(* IEC 61131-3 sources: std_i2980_v2.06_cp053/Source/IMM/ieccontrol/AutoCalibration1 (part 4) *)

GO_ON_TRANSITION TResetCalibBwd (* TResetCalibBwd *) FROM S_StopCalibBwd TO S_RESET :=  #BEGIN_EDIT_BLOCK
TRUE
;#END_EDIT_BLOCK
END_TRANSITION

TRANSITION TStartWriteBwd (* TStartWriteBwd *) FROM S_CHECK_ALARMS_BWD TO S_WRITE_BWD :=  #BEGIN_EDIT_BLOCK
S_CHECK_ALARMS_BWD.T > T#100ms
;#END_EDIT_BLOCK
END_TRANSITION

GO_ON_TRANSITION TStopIdentBwd2 (* TStopCalibBwd2 *) FROM S_CHECK_ALARMS_BWD TO S_StopCalibBwd :=  #BEGIN_EDIT_BLOCK
sv_iPendingAlarms <> 0
;#END_EDIT_BLOCK
END_TRANSITION

TRANSITION TWriteBwd (* TWriteBwd *) FROM S_WRITE_BWD TO S_CHECK_MINSPEED_BWD :=  #BEGIN_EDIT_BLOCK
mbLogFileSaved
;#END_EDIT_BLOCK
END_TRANSITION

TRANSITION TMaxBwdDetected (* TMaxBwdDetected *) FROM S_CHECK_MINSPEED_BWD TO S_MoveEndBwd :=  #BEGIN_EDIT_BLOCK
bMinBwdDetected
;#END_EDIT_BLOCK
END_TRANSITION

TRANSITION TMaxBwdRetry (* TMaxBwdRetry *) FROM S_CHECK_MINSPEED_BWD TO S_ReadyMinBwdRetry :=  #BEGIN_EDIT_BLOCK
bMinBwdRetry
;#END_EDIT_BLOCK
END_TRANSITION

TRANSITION TReadyMinBwdRetry (* Trans49 *) FROM S_ReadyMinBwdRetry TO S_MinBwdRetry :=  #BEGIN_EDIT_BLOCK
fbCheckReady.bReady
;#END_EDIT_BLOCK
END_TRANSITION

TRANSITION TMoveFwdDone (* TMoveFwdDone *) FROM S_MinBwdRetry TO S_CHECK_ALARMS_RETRYBWD :=  #BEGIN_EDIT_BLOCK
bMoveFwdDone
;#END_EDIT_BLOCK
END_TRANSITION

GO_ON_TRANSITION TStopMoveFwd (* TStopMoveFwd *) FROM S_MinBwdRetry TO S_StopMoveFwd :=  #BEGIN_EDIT_BLOCK
sv_GlobalIdentMinSpeedStatus.Status = tnCalibState_Aborted OR
sv_GlobalIdentMinSpeedStatus.Status = tnCalibState_None
OR sv_iPendingAlarms <> 0
OR mActMovement^.bRedo = FALSE

;#END_EDIT_BLOCK
END_TRANSITION

TRANSITION TResetBwd (* TResetBwd *) FROM S_StopMoveFwd TO S_RESET :=  #BEGIN_EDIT_BLOCK
TRUE
;#END_EDIT_BLOCK
END_TRANSITION

TRANSITION TRetryBwd (* TRetryBwd *) FROM S_CHECK_ALARMS_RETRYBWD TO S_CALIB_BWD :=  #BEGIN_EDIT_BLOCK
S_CHECK_ALARMS_RETRYBWD.T > T#1s
;#END_EDIT_BLOCK
END_TRANSITION

GO_ON_TRANSITION TStopIdentBwd4 (* TStopIdentBwd4 *) FROM S_CHECK_ALARMS_RETRYBWD TO S_StopMoveFwd :=  #BEGIN_EDIT_BLOCK
sv_iPendingAlarms <> 0
;#END_EDIT_BLOCK
END_TRANSITION

TRANSITION TMoveEndBwdDone (* TMoveEndBwdDone *) FROM S_MoveEndBwd TO S_Done :=  #BEGIN_EDIT_BLOCK
bMoveBwdDone
;#END_EDIT_BLOCK
END_TRANSITION

GO_ON_TRANSITION TStopMoveEndBwd (* TStopMoveEndBwd *) FROM S_MoveEndBwd TO S_StopMoveEndBwd :=  #BEGIN_EDIT_BLOCK
sv_GlobalIdentMinSpeedStatus.Status = tnCalibState_Aborted OR
sv_GlobalIdentMinSpeedStatus.Status = tnCalibState_None
OR sv_iPendingAlarms <> 0
;#END_EDIT_BLOCK
END_TRANSITION

GO_ON_TRANSITION TResetMoveEndBwd (* TResetMoveEndBwd *) FROM S_StopMoveEndBwd TO S_RESET :=  #BEGIN_EDIT_BLOCK
TRUE
;#END_EDIT_BLOCK
END_TRANSITION

TRANSITION TDone (* TDone *) FROM S_Done TO S_RESET :=  #BEGIN_EDIT_BLOCK
TRUE
;#END_EDIT_BLOCK
END_TRANSITION

(* end IecGraph-Code *)
(* sfc-code *)
(* end sfc-code *)

END_ALGORITHM

POSTUPDATE_ALGORITHM pMinCommandListen ON PU_Task_7 WITH sv_GlobalIdentMinSpeedStatus.Command,sv_GlobalIdentMinSpeedStatus.bStart

VAR_TEMP
 i : DINT;
END_VAR
#BEGIN_EDIT_BLOCK
//stop all calibrations
// TEST
IF sv_GlobalIdentMinSpeedStatus.Command = tnCalibCommand_Stop THEN
    sv_GlobalIdentMinSpeedStatus.bStart := FALSE;
END_IF;
//
IF sv_GlobalIdentMinSpeedStatus.Command = tnCalibCommand_Stop OR (NOT sv_GlobalIdentMinSpeedStatus.bStart) THEN
    FOR i:= 1 TO cCalibMovements DO
        IF CHECK_REF(sv_GlobalIdentMinSpeedStatus.pMovements[i]^) THEN
            IF sv_GlobalIdentMinSpeedStatus.pMovements[i]^.Status = tnCalibState_Running OR
               sv_GlobalIdentMinSpeedStatus.pMovements[i]^.bRedo THEN
                sv_GlobalIdentMinSpeedStatus.pMovements[i]^.Status := tnCalibState_Aborted;
                sv_GlobalIdentMinSpeedStatus.pMovements[i]^.bRedo := FALSE;//FIXME: check if needed
                sv_GlobalIdentMinSpeedStatus.Status := tnCalibState_Aborted;
                EXIT;
            END_IF;
        END_IF;
    END_FOR;
    IF (sv_GlobalIdentMinSpeedStatus.Command = tnCalibCommand_Stop) THEN
       IF (sv_GlobalIdentMinSpeedStatus.Status <> tnCalibState_Aborted) THEN
          sv_GlobalIdentMinSpeedStatus.Status := tnCalibState_None;
       END_IF;

    END_IF;
ELSIF (sv_GlobalIdentMinSpeedStatus.Command = tnCalibCommand_Start) OR (sv_GlobalIdentMinSpeedStatus.bStart) THEN
    IF sv_OperationMode = nSetup THEN
        mbUseSingleMovement := FALSE;
        START_PROCESS_ALGORITHM(paMinCalibSequence);
    ELSE
        sv_GlobalIdentMinSpeedStatus.bStart := FALSE;
        SET_ALARM(erSetupModeRequiredForCalib);
    END_IF;
END_IF;
sv_GlobalIdentMinSpeedStatus.Command := tnCalibCommand_None;

;#END_EDIT_BLOCK END_ALGORITHM

(*
Coordinate sequential start of auto calib cycle
starts one auto calib movement after the other
*)

PROCESS_ALGORITHM paMinCalibSequence ON TaskMid

VAR_TEMP
 j : DINT;
 i : DINT;
END_VAR

VAR
 tmpMovements : tyIdentSpeedMovements;
 iMaxMovements : DINT;
 tmpM : tpIdentSpeedMovement;
 ConstBwdVis : tsVelPre;
END_VAR

(* IecGraph-Code *)

(* init step *)
INITIAL_STEP S_INIT:
ASortCalibs (P);
Action108 (P);
END_STEP

ACTION ASortCalibs: #BEGIN_EDIT_BLOCK
sv_GlobalIdentMinSpeedStatus.Status := tnCalibState_Running;
miErrorNo := 0;

tmpMovements := sv_GlobalIdentMinSpeedStatus.pMovements;

(* get number of movements *)
FOR i:= 1 TO cCalibMovements DO
    IF NOT CHECK_REF(tmpMovements[i]^)  THEN
        EXIT;
    END_IF;
END_FOR;
iMaxMovements := i -1;

(* sort them by iOrder *)
FOR i := 1 TO iMaxMovements -1 DO
    FOR j := 1 TO iMaxMovements - 1 - i +1 DO
        IF tmpMovements[j]^.iOrder > tmpMovements[j + 1]^.iOrder THEN
            tmpM := tmpMovements[j];
            tmpMovements[j] := tmpMovements[j + 1];
            tmpMovements[j + 1] := tmpM;
        END_IF;
    END_FOR;
END_FOR;

;#END_EDIT_BLOCK END_ACTION (*ASortCalibs*)
ACTION Action108: #BEGIN_EDIT_BLOCK
mCalibCounter := 0;
sv_GlobalIdentMinSpeedStatus.iCurrentStep := mCalibCounter;

;#END_EDIT_BLOCK END_ACTION (*Action108*)

(* steps *)
STEP S_RESET:
AReset (P);
AStopMovements (N);
AStopSelf (P);
END_STEP

ACTION AReset: #BEGIN_EDIT_BLOCK
sv_bAutoIdentRunning := FALSE;

;#END_EDIT_BLOCK END_ACTION (*AReset*)
ACTION AStopMovements: #BEGIN_EDIT_BLOCK
(* stop all identification movements *)
FOR i:= 1 TO cCalibMovements DO
    IF CHECK_REF(sv_GlobalIdentMinSpeedStatus.pMovements[i]^) THEN
        IF sv_GlobalIdentMinSpeedStatus.pMovements[i]^.Status = tnCalibState_Running OR
           sv_GlobalIdentMinSpeedStatus.pMovements[i]^.bRedo THEN
            sv_GlobalIdentMinSpeedStatus.pMovements[i]^.Status := tnCalibState_Aborted;
            sv_GlobalIdentMinSpeedStatus.pMovements[i]^.bRedo := FALSE;//FIXME: check if needed
            EXIT;
        END_IF;
    END_IF;
END_FOR;

;#END_EDIT_BLOCK END_ACTION (*AStopMovements*)
ACTION AStopSelf: #BEGIN_EDIT_BLOCK
sv_GlobalIdentMinSpeedStatus.bStart := FALSE;
STOP_PROCESS_ALGORITHM();

;#END_EDIT_BLOCK END_ACTION (*AStopSelf*)
STEP Step74:
AAnyCoreActive (N);
END_STEP

STEP Step19:
ASignalStart (P);
END_STEP

ACTION ASignalStart: #BEGIN_EDIT_BLOCK
sv_bAutoIdentRunning := TRUE;

;#END_EDIT_BLOCK END_ACTION (*ASignalStart*)
STEP S_MoveEjectorBack:
AEjectorBack (P);
Action116 (N);
AResetEjectorBack (P0);
END_STEP

ACTION Action116: #BEGIN_EDIT_BLOCK
fbCheckReady(DeviceId := DeviceIdEjector)

;#END_EDIT_BLOCK END_ACTION (*Action116*)
ACTION AResetEjectorBack: #BEGIN_EDIT_BLOCK
miErrorNo := 0;
sv_EjectorIdentMinMovement.prIdentPosition^ := 0.0;
sv_EjectorIdentMinMovement.prStopRamp^ := 0.0;
sv_EjectorIdentMinMovement.pbMoveIdent^ := FALSE;
sv_EjectorIdentMinMovement.pConstBwdVis^ := ConstBwdVis;

;#END_EDIT_BLOCK END_ACTION (*AResetEjectorBack*)
STEP S_StopEjector:
AStopEjeMovement (P);
END_STEP

STEP S_MoveMoldBack:
AMoldBack (P);
Action118 (N);
AResetMoldBack (P0);
END_STEP

ACTION Action118: #BEGIN_EDIT_BLOCK
fbCheckReady(DeviceId := DeviceIdMold)

;#END_EDIT_BLOCK END_ACTION (*Action118*)
ACTION AResetMoldBack: #BEGIN_EDIT_BLOCK
miErrorNo := 0;
sv_MoldIdentMinMovement.prIdentPosition^ := 0.0;
sv_MoldIdentMinMovement.prStopRamp^ := 0.0;
sv_MoldIdentMinMovement.pbMoveIdent^ := FALSE;
sv_MoldIdentMinMovement.pConstBwdVis^ := ConstBwdVis;

;#END_EDIT_BLOCK END_ACTION (*AResetMoldBack*)
STEP S_StopMold:
AStopMoldMovement (P);
END_STEP

STEP S_CALIB_SINGLE:
AStartMovementStart (P);
END_STEP

ACTION AStartMovementStart: #BEGIN_EDIT_BLOCK
IF mCalibCounter < iMaxMovements THEN
   mCalibCounter := mCalibCounter +1;
   tmpMovements[mCalibCounter]^.bRedo := TRUE;
END_IF;

;#END_EDIT_BLOCK END_ACTION (*AStartMovementStart*)
STEP S_CHECKNEXT:
END_STEP

STEP S_StopIdent:
AStopIdent (P);
END_STEP

ACTION AStopIdent: #BEGIN_EDIT_BLOCK
sv_GlobalIdentMinSpeedStatus.Status := tnCalibState_Done;

;#END_EDIT_BLOCK END_ACTION (*AStopIdent*)

(* transitions *)
TRANSITION Trans50 (* Trans50 *) FROM S_RESET TO S_INIT :=  #BEGIN_EDIT_BLOCK
TRUE
;#END_EDIT_BLOCK
END_TRANSITION

TRANSITION Trans80 (* Trans80 *) FROM S_INIT TO Step19 :=  #BEGIN_EDIT_BLOCK
NOT sv_bCoresActive AND
sv_iPendingAlarms = 0
;#END_EDIT_BLOCK
(*Comment : Start with moving ejector and
mold in backward position, check if any failure
occured.
After that start the calibration cycle, if no alarm is
pending*)
END_TRANSITION

GO_ON_TRANSITION Trans87 (* Trans87 *) FROM S_INIT TO Step74 :=  #BEGIN_EDIT_BLOCK
sv_bCoresActive OR
sv_iPendingAlarms > 0

;#END_EDIT_BLOCK
END_TRANSITION

TRANSITION Trans88 (* Trans88 *) FROM Step74 TO S_RESET :=  #BEGIN_EDIT_BLOCK
TRUE

;#END_EDIT_BLOCK
END_TRANSITION

TRANSITION Trans18 (* Trans18 *) FROM Step19 TO S_MoveEjectorBack :=  #BEGIN_EDIT_BLOCK
TRUE
;#END_EDIT_BLOCK
END_TRANSITION

TRANSITION Trans72 (* Trans72 *) FROM S_MoveEjectorBack TO S_MoveMoldBack :=  #BEGIN_EDIT_BLOCK
fbCheckReady.bReady AND
sv_iPendingAlarms = 0
;#END_EDIT_BLOCK
END_TRANSITION

GO_ON_TRANSITION Trans83 (* Trans83 *) FROM S_MoveEjectorBack TO S_StopEjector :=  #BEGIN_EDIT_BLOCK
sv_GlobalIdentMinSpeedStatus.Status = tnCalibState_Aborted OR
sv_GlobalIdentMinSpeedStatus.Status = tnCalibState_None
OR sv_iPendingAlarms <> 0
;#END_EDIT_BLOCK
END_TRANSITION

TRANSITION Trans84 (* Trans84 *) FROM S_StopEjector TO S_RESET :=  #BEGIN_EDIT_BLOCK
TRUE

;#END_EDIT_BLOCK
END_TRANSITION

TRANSITION Trans81 (* Trans81 *) FROM S_MoveMoldBack TO S_CALIB_SINGLE :=  #BEGIN_EDIT_BLOCK
fbCheckReady.bReady AND
sv_iPendingAlarms = 0
;#END_EDIT_BLOCK
END_TRANSITION

GO_ON_TRANSITION Trans85 (* Trans85 *) FROM S_MoveMoldBack TO S_StopMold :=  #BEGIN_EDIT_BLOCK
sv_GlobalIdentMinSpeedStatus.Status = tnCalibState_Aborted OR
sv_GlobalIdentMinSpeedStatus.Status = tnCalibState_None
OR sv_iPendingAlarms <> 0
;#END_EDIT_BLOCK
END_TRANSITION

TRANSITION Trans86 (* Trans86 *) FROM S_StopMold TO S_RESET :=  #BEGIN_EDIT_BLOCK
TRUE
;#END_EDIT_BLOCK
END_TRANSITION

TRANSITION TCheckActMoveReady (* TCheckActMoveReady *) FROM S_CALIB_SINGLE TO S_CHECKNEXT :=  #BEGIN_EDIT_BLOCK
tmpMovements[mCalibCounter]^.bRedo = FALSE AND
NOT(sv_GlobalIdentMinSpeedStatus.Status = tnCalibState_Aborted OR
    sv_GlobalIdentMinSpeedStatus.Status = tnCalibState_Error)
;#END_EDIT_BLOCK
END_TRANSITION

GO_ON_TRANSITION TCheckError (* TCheckError *) FROM S_CALIB_SINGLE TO S_RESET :=  #BEGIN_EDIT_BLOCK
sv_GlobalIdentMinSpeedStatus.Status = tnCalibState_Aborted OR
sv_GlobalIdentMinSpeedStatus.Status = tnCalibState_Error OR
iMaxMovements = 0
;#END_EDIT_BLOCK
END_TRANSITION

TRANSITION TNextUnit (* TNextUnit *) FROM S_CHECKNEXT TO S_CALIB_SINGLE :=  #BEGIN_EDIT_BLOCK
mCalibCounter < iMaxMovements
//AND S_CHECKNEXT.T>T#3s
;#END_EDIT_BLOCK
END_TRANSITION

TRANSITION TStopIdent (* TStopIdent *) FROM S_CHECKNEXT TO S_StopIdent :=  #BEGIN_EDIT_BLOCK
mCalibCounter >= iMaxMovements
;#END_EDIT_BLOCK
END_TRANSITION

TRANSITION TReset (* TReset *) FROM S_StopIdent TO S_RESET :=  #BEGIN_EDIT_BLOCK
TRUE
;#END_EDIT_BLOCK
END_TRANSITION

(* end IecGraph-Code *)
(* sfc-code *)

(* stand alone actions *)
ACTION AEjectorBack: #BEGIN_EDIT_BLOCK
miErrorNo := cIdentSpeedMinSequence;

IF sv_EjectorIdentMinMovement.bPositionIncreasingFwd THEN
   sv_EjectorIdentMinMovement.prIdentPosition^ := mrBwdStopPosition;
ELSE
   sv_EjectorIdentMinMovement.prIdentPosition^ := sv_EjectorIdentMinMovement.prStroke^ - mrBwdStopPosition;
END_IF;
sv_EjectorIdentMinMovement.prStopRamp^ := 1.0e10;
ConstBwdVis := sv_EjectorIdentMinMovement.pConstBwdVis^;
sv_EjectorIdentMinMovement.pConstBwdVis^.Pressure.Output.rRamp := MAX(1.0e10, sv_EjectorIdentMinMovement.pConstBwdVis^.Pressure.Output.rRamp);
sv_EjectorIdentMinMovement.pConstBwdVis^.Pressure.rMinOutput := 0.1 * sv_EjectorIdentMinMovement.prMaxPressureBwd^;
sv_EjectorIdentMinMovement.pbMoveIdent^ := TRUE;

evStartRequestData.DeviceId := DeviceIdEjector;
evStartRequestData.MoveDir := cMoveBwd;
evStartRequestData.MoveId := cMoveBwd;
SET_EVENT(evStartRequest, evStartRequestData);

;#END_EDIT_BLOCK END_ACTION (*AEjectorBack*)
ACTION AMoldBack: #BEGIN_EDIT_BLOCK
miErrorNo := cIdentSpeedMinSequence;

IF sv_MoldIdentMinMovement.bPositionIncreasingFwd THEN
   sv_MoldIdentMinMovement.prIdentPosition^ := mrBwdStopPosition;
ELSE
   sv_MoldIdentMinMovement.prIdentPosition^ := sv_MoldIdentMinMovement.prStroke^ - mrBwdStopPosition;
END_IF;
sv_MoldIdentMinMovement.prStopRamp^ := 1.0e10;
ConstBwdVis := sv_MoldIdentMinMovement.pConstBwdVis^;
sv_MoldIdentMinMovement.pConstBwdVis^.Pressure.Output.rRamp := MAX(1.0e10, sv_MoldIdentMinMovement.pConstBwdVis^.Pressure.Output.rRamp);
sv_MoldIdentMinMovement.pConstBwdVis^.Pressure.rMinOutput := 0.1 * sv_MoldIdentMinMovement.prMaxPressureBwd^;
sv_MoldIdentMinMovement.pbMoveIdent^ := TRUE;

evStartRequestData.DeviceId := DeviceIdMold;
evStartRequestData.MoveDir := cMoveBwd;
evStartRequestData.MoveId := cMoveBwd;
SET_EVENT(evStartRequest, evStartRequestData);

;#END_EDIT_BLOCK END_ACTION (*AMoldBack*)
ACTION AStopEjeMovement: #BEGIN_EDIT_BLOCK
evStopRequestData.DeviceId := DeviceIdEjector;
evStopRequestData.MoveDir := cMoveBwd;
evStopRequestData.MoveId := cMoveBwd;
SET_EVENT(evStopRequest, evStopRequestData);
IF sv_GlobalIdentMinSpeedStatus.Status <> tnCalibState_None THEN
    sv_GlobalIdentMinSpeedStatus.Status := tnCalibState_Aborted;
END_IF;

;#END_EDIT_BLOCK END_ACTION (*AStopEjeMovement*)
ACTION AStopMoldMovement: #BEGIN_EDIT_BLOCK
evStopRequestData.DeviceId := DeviceIdMold;
evStopRequestData.MoveDir := cMoveBwd;
evStopRequestData.MoveId := cMoveBwd;
SET_EVENT(evStopRequest, evStopRequestData);
IF sv_GlobalIdentMinSpeedStatus.Status <> tnCalibState_None THEN
    sv_GlobalIdentMinSpeedStatus.Status := tnCalibState_Aborted;
END_IF;

;#END_EDIT_BLOCK END_ACTION (*AStopMoldMovement*)
ACTION AAnyCoreActive: #BEGIN_EDIT_BLOCK
IF sv_bCoresActive THEN
   SET_ALARM(erCalibCoresActive);
END_IF;
sv_GlobalIdentMinSpeedStatus.Status := tnCalibState_Aborted;

;#END_EDIT_BLOCK END_ACTION (*AAnyCoreActive*)

(* exits *)

EXIT_TRANSITION E_NotSetupMode := #BEGIN_EDIT_BLOCK
sv_OperationMode <> nSetup
;#END_EDIT_BLOCK
PRIORITY 1 WITH  INITIAL_STEP S_RESET: END_STEP
END_TRANSITION
(* end sfc-code *)

END_ALGORITHM

POSTUPDATE_ALGORITHM pDataState ON PU_Task_13 WITH sv_DataState

VAR_TEMP
 i : DINT;
END_VAR

VAR
 bMDLoadingInProgress : BOOL (* loading of machine data in progress *);
END_VAR
#BEGIN_EDIT_BLOCK
(**************************************** WARNING ********************************************
 *** The KEBA Kemro K2 System including software is not intended for safety control tasks! ***
 ***                       For further information see Comment tab!                        ***
 *********************************************************************************************)

//reset calib state after loading machine data

IF sv_DataState = nReadMachineData THEN
   //loading of machinedata in progress
   bMDLoadingInProgress := TRUE;
   RETURN;
END_IF;

IF sv_DataState = nReady AND bMDLoadingInProgress THEN
   FOR i := 1 TO sv_GlobalIdentMaxSpeedStatus.iMaxStep DO
      //set state to tnCalibState_None
      sv_GlobalIdentMaxSpeedStatus.pMovements[i]^.Status := tnCalibState_None;
   END_FOR;
   FOR i := 1 TO sv_GlobalIdentMinSpeedStatus.iMaxStep DO
      //set state to tnCalibState_None
      sv_GlobalIdentMinSpeedStatus.pMovements[i]^.Status := tnCalibState_None;
   END_FOR;
   bMDLoadingInProgress := FALSE;
END_IF;

;#END_EDIT_BLOCK END_ALGORITHM

END_ALGORITHM_BLOCK

#END_OF_IEC_PART

@Puma @IecEditor 6 152 @Pou 25
@@@BEG_Comment@@@

@@@END_Comment@@@

@BEG_Contents

@BEG_Func
@RT(17)FuncTreeContainer
4
@Var @RT(14)GET_SYNC_REFTO @RT(0) @T @T @DERIVED 0 @F @RT(22)KEBA_STANDARD_FUNCTION @F
@T
@BEG_Attrib
0 @RT(0) @RT(0)
@END_Attrib
1 1 @F @F @F @F

@Var @RT(9)SET_ALARM @RT(0) @T @T @DERIVED 0 @F @RT(23)KEBA_STANDARD_PROCEDURE @F
@T
@BEG_Attrib
0 @RT(0) @RT(0)
@END_Attrib
1 1 @F @F @F @F

@Var @RT(9)SET_EVENT @RT(0) @T @T @DERIVED 0 @F @RT(23)KEBA_STANDARD_PROCEDURE @F
@T
@BEG_Attrib
0 @RT(0) @RT(0)
@END_Attrib
1 1 @F @F @F @F

@Var @RT(9)CHECK_REF @RT(0) @T @T @DERIVED 0 @F @RT(23)KEBA_STANDARD_PROCEDURE @F
@T
@BEG_Attrib
0 @RT(0) @RT(0)
@END_Attrib
1 1 @F @F @F @F

@END_Func

@BEG_Const
@RT(18)ConstTreeContainer
18
@Var @RT(12)cCompEjector @RT(0) @T @F @DT @RT(4)DINT @RT(0) @T @T @BASIC 0 @F
@F @F
@T
@BEG_Attrib
0 @RT(3)102 @RT(17)Component Ejector
@END_Attrib
1 1 @F @F @F @F

@Var @RT(9)cCompMold @RT(0) @T @F @DT @RT(4)DINT @RT(0) @T @T @BASIC 0 @F
@F @F
@T
@BEG_Attrib
0 @RT(3)101 @RT(14)Component Mold
@END_Attrib
1 1 @F @F @F @F

@Var @RT(14)KSYS_Status_OK @RT(0) @T @T @DERIVED 0 @F @RT(11)KSYS_Status @F
@T
@BEG_Attrib
0 @RT(1)1 @RT(0)
@END_Attrib
1 1 @F @F @F @F

@Var @RT(16)cOptionHydraulic @RT(0) @T @F @DT @RT(5)DWORD @RT(0) @T @T @BASIC 0 @F
@F @F
@T
@BEG_Attrib
0 @RT(5)16#01 @RT(26)Hydraulic device, LSB is 1
@END_Attrib
1 1 @F @F @F @F

@Var @RT(17)tnCalibState_None @RT(0) @T @T @DERIVED 0 @F @RT(12)tnCalibState @F
@T
@BEG_Attrib
0 @RT(1)0 @RT(0)
@END_Attrib
1 1 @F @F @F @F

@Var @RT(20)tnCalibState_Running @RT(0) @T @T @DERIVED 0 @F @RT(12)tnCalibState @F
@T
@BEG_Attrib
0 @RT(1)1 @RT(23)calibration in progress
@END_Attrib
1 1 @F @F @F @F

@Var @RT(19)tnCalibCommand_Stop @RT(0) @T @T @DERIVED 0 @F @RT(14)tnCalibCommand @F
@T
@BEG_Attrib
0 @RT(1)2 @RT(0)
@END_Attrib
1 1 @F @F @F @F

@Var @RT(20)tnCalibState_Aborted @RT(0) @T @T @DERIVED 0 @F @RT(12)tnCalibState @F
@T
@BEG_Attrib
0 @RT(1)4 @RT(19)calibration aborted
@END_Attrib
1 1 @F @F @F @F

@Var @RT(8)cMoveFwd @RT(0) @T @F @DT @RT(4)DINT @RT(0) @T @T @BASIC 0 @F
@F @F
@T
@BEG_Attrib
0 @RT(2)12 @RT(16)movement forward
@END_Attrib
1 1 @F @F @F @F

@Var @RT(9)cMoveNone @RT(0) @T @F @DT @RT(4)DINT @RT(0) @T @T @BASIC 0 @F
@F @F
@T
@BEG_Attrib
0 @RT(13)cMinMoveIdent @RT(4)None
@END_Attrib
1 1 @F @F @F @F

@Var @RT(8)cMoveBwd @RT(0) @T @F @DT @RT(4)DINT @RT(0) @T @T @BASIC 0 @F
@F @F
@T
@BEG_Attrib
0 @RT(2)11 @RT(17)movement backward
@END_Attrib
1 1 @F @F @F @F

@Var @RT(19)cMoveDecompAftPlast @RT(0) @T @F @DT @RT(4)DINT @RT(0) @T @T @BASIC 0 @F
@F @F
@T
@BEG_Attrib
0 @RT(2)27 @RT(25)decompression after plast
@END_Attrib
1 1 @F @F @F @F

@Var @RT(18)tnCalibState_Error @RT(0) @T @T @DERIVED 0 @F @RT(12)tnCalibState @F
@T
@BEG_Attrib
0 @RT(1)3 @RT(32)error occured during calibration
@END_Attrib
1 1 @F @F @F @F

@Var @RT(15)cCalibMovements @RT(0) @T @F @DT @RT(4)DINT @RT(0) @T @T @BASIC 0 @F
@F @F
@T
@BEG_Attrib
0 @RT(2)30 @RT(0)
@END_Attrib
1 1 @F @F @F @F

@Var @RT(6)nSetup @RT(0) @T @T @DERIVED 0 @F @RT(15)tnOperationMode @F
@T
@BEG_Attrib
0 @RT(1)0 @RT(36)Setup mode only for service engineer
@END_Attrib
1 1 @F @F @F @F

@Var @RT(19)tnCalibCommand_None @RT(0) @T @T @DERIVED 0 @F @RT(14)tnCalibCommand @F
@T
@BEG_Attrib
0 @RT(1)0 @RT(0)
@END_Attrib
1 1 @F @F @F @F

@Var @RT(17)tnCalibState_Done @RT(0) @T @T @DERIVED 0 @F @RT(12)tnCalibState @F
@T
@BEG_Attrib
0 @RT(1)2 @RT(33)calibration finished successfully
@END_Attrib
1 1 @F @F @F @F

@Var @RT(20)tnCalibCommand_Start @RT(0) @T @T @DERIVED 0 @F @RT(14)tnCalibCommand @F
@T
@BEG_Attrib
0 @RT(1)1 @RT(0)
@END_Attrib
1 1 @F @F @F @F

@END_Const

@BEG_Export

@BEG_Kind
@ALGORITHM_BLOCK @RT(16)ABAutoIdentSpeed @STRUCTURED_TEXT
@RT(0) @RT(0) @RT(0)
@END_Kind

@BEG_Dcl
@RT(16)DclTreeContainer
76
@Var @RT(28)sv_GlobalIdentMaxSpeedStatus @RT(0) @T @T @DERIVED 0 @T @T @DT @RT(24)tsGlobalIdentSpeedStatus @RT(0) @T @T @UNKNOWN 0 @F
@F @F
@T
@BEG_Attrib
3 @RT(0) @RT(0) @RT(0)
@END_Attrib
1 8 @F @F @F @F

@Var @RT(26)sv_EjectorIdentMaxMovement @RT(0) @T @T @DERIVED 0 @T @T @DT @RT(20)tsIdentSpeedMovement @RT(0) @T @T @UNKNOWN 0 @F
@F @F
@T
@BEG_Attrib
3 @RT(0) @RT(0) @RT(0)
@END_Attrib
1 8 @F @F @F @F

@Var @RT(23)sv_MoldIdentMaxMovement @RT(0) @T @T @DERIVED 0 @T @T @DT @RT(20)tsIdentSpeedMovement @RT(0) @T @T @UNKNOWN 0 @F
@F @F
@T
@BEG_Attrib
3 @RT(0) @RT(0) @RT(0)
@END_Attrib
1 8 @F @F @F @F

@Var @RT(28)sv_InjectionIdentMaxMovement @RT(0) @T @T @DERIVED 0 @T @T @DT @RT(20)tsIdentSpeedMovement @RT(0) @T @T @UNKNOWN 0 @F
@F @F
@T
@BEG_Attrib
3 @RT(0) @RT(0) @RT(0)
@END_Attrib
1 8 @F @F @F @F

@Var @RT(25)sv_NozzleIdentMaxMovement @RT(0) @T @T @DERIVED 0 @T @T @DT @RT(20)tsIdentSpeedMovement @RT(0) @T @T @UNKNOWN 0 @F
@F @F
@T
@BEG_Attrib
3 @RT(0) @RT(0) @RT(0)
@END_Attrib
1 8 @F @F @F @F

@Var @RT(28)sv_GlobalIdentMinSpeedStatus @RT(0) @T @T @DERIVED 0 @T @T @DT @RT(24)tsGlobalIdentSpeedStatus @RT(0) @T @T @UNKNOWN 0 @F
@F @F
@T
@BEG_Attrib
3 @RT(0) @RT(0) @RT(0)
@END_Attrib
1 8 @F @F @F @F

@Var @RT(26)sv_EjectorIdentMinMovement @RT(0) @T @T @DERIVED 0 @T @T @DT @RT(20)tsIdentSpeedMovement @RT(0) @T @T @UNKNOWN 0 @F
@F @F
@T
@BEG_Attrib
3 @RT(0) @RT(0) @RT(0)
@END_Attrib
1 8 @F @F @F @F

@Var @RT(23)sv_MoldIdentMinMovement @RT(0) @T @T @DERIVED 0 @T @T @DT @RT(20)tsIdentSpeedMovement @RT(0) @T @T @UNKNOWN 0 @F
@F @F
@T
@BEG_Attrib
3 @RT(0) @RT(0) @RT(0)
@END_Attrib
1 8 @F @F @F @F

@Var @RT(28)sv_InjectionIdentMinMovement @RT(0) @T @T @DERIVED 0 @T @T @DT @RT(20)tsIdentSpeedMovement @RT(0) @T @T @UNKNOWN 0 @F
@F @F
@T
@BEG_Attrib
3 @RT(0) @RT(0) @RT(0)
@END_Attrib
1 8 @F @F @F @F

@Var @RT(25)sv_NozzleIdentMinMovement @RT(0) @T @T @DERIVED 0 @T @T @DT @RT(20)tsIdentSpeedMovement @RT(0) @T @T @UNKNOWN 0 @F
@F @F
@T
@BEG_Attrib
3 @RT(0) @RT(0) @RT(0)
@END_Attrib
1 8 @F @F @F @F

@Var @RT(17)sv_iPendingAlarms @RT(0) @T @F @DT @RT(4)DINT @RT(0) @T @T @BASIC 0 @F
@F @F
@T
@BEG_Attrib
3 @RT(0) @RT(0) @RT(0)
@END_Attrib
1 8 @F @F @F @F

@Var @RT(16)sv_OperationMode @RT(0) @T @T @DERIVED 0 @T @T @DT @RT(15)tnOperationMode @RT(0) @T @T @UNKNOWN 0 @F
@F @F
@T
@BEG_Attrib
3 @RT(0) @RT(0) @RT(0)
@END_Attrib
1 8 @F @F @F @F

@Var @RT(20)sv_bAutoIdentRunning @RT(0) @T @F @DT @RT(4)BOOL @RT(0) @T @T @BASIC 0 @F
@F @F
@T
@BEG_Attrib
3 @RT(0) @RT(23)auto calibration active @RT(0)
@END_Attrib
1 8 @F @F @F @F

@Var @RT(15)sv_bCoresActive @RT(0) @T @F @DT @RT(4)BOOL @RT(0) @T @T @BASIC 0 @F
@F @F
@T
@BEG_Attrib
3 @RT(0) @RT(0) @RT(0)
@END_Attrib
1 8 @F @F @F @F

@Var @RT(11)sv_PumpData @RT(0) @T @T @DERIVED 0 @T @T @DT @RT(10)tyPumpData @RT(0) @T @T @UNKNOWN 0 @F
@F @F
@T
@BEG_Attrib
3 @RT(0) @RT(0) @RT(0)
@END_Attrib
1 8 @F @F @F @F

@Var @RT(7)TaskMid @RT(0) @T @F @DT @RT(4)TASK @RT(0) @T @T @BASIC 0 @F
@F @F
@T
@BEG_Attrib
3 @RT(0) @RT(0) @RT(0)
@END_Attrib
1 7 @F @F @F @F

@Var @RT(8)TaskSlow @RT(0) @T @F @DT @RT(4)TASK @RT(0) @T @T @BASIC 0 @F
@F @F
@T
@BEG_Attrib
3 @RT(0) @RT(0) @RT(0)
@END_Attrib
1 7 @F @F @F @F

@Var @RT(10)TaskInject @RT(0) @T @F @DT @RT(4)TASK @RT(0) @T @T @BASIC 0 @F
@F @F
@T
@BEG_Attrib
3 @RT(0) @RT(0) @RT(0)
@END_Attrib
1 7 @F @F @F @F

@Var @RT(10)TaskAnalog @RT(0) @T @F @DT @RT(4)TASK @RT(0) @T @T @BASIC 0 @F
@F @F
@T
@BEG_Attrib
3 @RT(0) @RT(0) @RT(0)
@END_Attrib
1 7 @F @F @F @F

@Var @RT(9)PU_Task_7 @RT(0) @T @F @DT @RT(4)TASK @RT(0) @T @T @BASIC 0 @F
@F @F
@T
@BEG_Attrib
3 @RT(0) @RT(0) @RT(0)
@END_Attrib
1 7 @F @F @F @F

@Var @RT(9)EV_Task_7 @RT(0) @T @F @DT @RT(4)TASK @RT(0) @T @T @BASIC 0 @F
@F @F
@T
@BEG_Attrib
3 @RT(0) @RT(0) @RT(0)
@END_Attrib
1 7 @F @F @F @F

@Var @RT(25)erCalibrationSpeedStopped @RT(0) @T @F @DT @RT(5)ALARM @RT(0) @T @T @BASIC 0 @F
@F @F
@T
@BEG_Attrib
3 @RT(0) @RT(0) @RT(0)
@END_Attrib
1 7 @F @F @F @F

@Var @RT(27)erSetupModeRequiredForCalib @RT(0) @T @F @DT @RT(5)ALARM @RT(0) @T @T @BASIC 0 @F
@F @F
@T
@BEG_Attrib
3 @RT(0) @RT(0) @RT(0)
@END_Attrib
1 7 @F @F @F @F

@Var @RT(18)erCalibCoresActive @RT(0) @T @F @DT @RT(5)ALARM @RT(0) @T @T @BASIC 0 @F
@F @F
@T
@BEG_Attrib
3 @RT(0) @RT(0) @RT(0)
@END_Attrib
1 7 @F @F @F @F

@Var @RT(24)evRedoIdentMaxSpeedStart @RT(0) @T @T @DERIVED 0 @T @T @DT @RT(22)tevRedoIdentSpeedEvent @RT(0) @T @T @UNKNOWN 0 @F
@F @F
@T
@BEG_Attrib
3 @RT(0) @RT(0) @RT(0)
@END_Attrib
1 7 @F @F @F @F

@Var @RT(24)evRedoIdentMinSpeedStart @RT(0) @T @T @DERIVED 0 @T @T @DT @RT(22)tevRedoIdentSpeedEvent @RT(0) @T @T @UNKNOWN 0 @F
@F @F
@T
@BEG_Attrib
3 @RT(0) @RT(0) @RT(0)
@END_Attrib
1 7 @F @F @F @F

@Var @RT(13)evStopRequest @RT(0) @T @T @DERIVED 0 @T @T @DT @RT(14)tevStopRequest @RT(0) @T @T @UNKNOWN 0 @F
@F @F
@T
@BEG_Attrib
3 @RT(0) @RT(0) @RT(0)
@END_Attrib
1 7 @F @F @F @F

@Var @RT(14)evStartRequest @RT(0) @T @T @DERIVED 0 @T @T @DT @RT(15)tevStartRequest @RT(0) @T @T @UNKNOWN 0 @F
@F @F
@T
@BEG_Attrib
3 @RT(0) @RT(0) @RT(0)
@END_Attrib
1 7 @F @F @F @F

@Var @RT(15)DeviceIdEjector @RT(0) @T @T @DERIVED 0 @T @T @DT @RT(10)tsDeviceId @RT(0) @T @T @UNKNOWN 0 @F
@F @F
@T
@BEG_Attrib
3 @RT(33)(CompId:=cCompEjector,IndexId:=1) @RT(0) @RT(0)
@END_Attrib
1 0 @F @F @F @F

@Var @RT(12)DeviceIdMold @RT(0) @T @T @DERIVED 0 @T @T @DT @RT(10)tsDeviceId @RT(0) @T @T @UNKNOWN 0 @F
@F @F
@T
@BEG_Attrib
3 @RT(30)(CompId:=cCompMold,IndexId:=1) @RT(0) @RT(0)
@END_Attrib
1 0 @F @F @F @F

@Var @RT(12)mActMovement @RT(0) @T @T @DERIVED 0 @T @T @DT @RT(20)tpIdentSpeedMovement @RT(0) @T @T @UNKNOWN 0 @F
@F @F
@T
@BEG_Attrib
3 @RT(0) @RT(0) @RT(0)
@END_Attrib
1 0 @F @F @F @F

@Var @RT(13)mCalibCounter @RT(0) @T @F @DT @RT(4)DINT @RT(0) @T @T @BASIC 0 @F
@F @F
@T
@BEG_Attrib
3 @RT(0) @RT(0) @RT(0)
@END_Attrib
1 0 @F @F @F @F

@Var @RT(19)mbUseSingleMovement @RT(0) @T @F @DT @RT(4)BOOL @RT(0) @T @T @BASIC 0 @F
@F @F
@T
@BEG_Attrib
3 @RT(0) @RT(0) @RT(0)
@END_Attrib
1 0 @F @F @F @F

@Var @RT(12)fbCheckReady @RT(0) @T @T @DERIVED 0 @T @T @DT @RT(12)FBCheckReady @RT(0) @T @T @UNKNOWN 0 @F
@F @F
@T
@BEG_Attrib
3 @RT(0) @RT(0) @RT(0)
@END_Attrib
1 0 @F @F @F @F

@Var @RT(18)evStartRequestData @RT(0) @T @T @DERIVED 0 @T @T @DT @RT(19)tevStartRequestData @RT(0) @T @T @UNKNOWN 0 @F
@F @F
@T
@BEG_Attrib
3 @RT(0) @RT(0) @RT(0)
@END_Attrib
1 0 @F @F @F @F

@Var @RT(17)evStopRequestData @RT(0) @T @T @DERIVED 0 @T @T @DT @RT(18)tevStopRequestData @RT(0) @T @T @UNKNOWN 0 @F
@F @F
@T
@BEG_Attrib
3 @RT(0) @RT(0) @RT(0)
@END_Attrib
1 0 @F @F @F @F

@Var @RT(15)fbIdentWriteLog @RT(0) @T @T @DERIVED 0 @T @T @DT @RT(20)FBIdentSpeedWriteLog @RT(0) @T @T @UNKNOWN 0 @F
@F @F
@T
@BEG_Attrib
3 @RT(0) @RT(0) @RT(0)
@END_Attrib
1 0 @F @F @F @F

@Var @RT(13)miFileCounter @RT(0) @T @F @DT @RT(5)UDINT @RT(0) @T @T @BASIC 0 @F
@F @F
@T
@BEG_Attrib
3 @RT(0) @RT(0) @RT(0)
@END_Attrib
1 0 @F @F @F @F

@Var @RT(13)mbDeleteFiles @RT(0) @T @F @DT @RT(4)BOOL @RT(0) @T @T @BASIC 0 @F
@F @F
@T
@BEG_Attrib
3 @RT(0) @RT(0) @RT(0)
@END_Attrib
1 0 @F @F @F @F

@Var @RT(14)mbLogFileSaved @RT(0) @T @F @DT @RT(4)BOOL @RT(0) @T @T @BASIC 0 @F
@F @F
@T
@BEG_Attrib
3 @RT(4)TRUE @RT(0) @RT(0)
@END_Attrib
1 0 @F @F @F @F

@Var @RT(10)msFileName @RT(0) @T @F @DT @RT(11)STRING(255) @RT(0) @T @T @STRING 0 @F @RT(3)255 @F
@F @F
@T
@BEG_Attrib
3 @RT(0) @RT(0) @RT(0)
@END_Attrib
1 0 @F @F @F @F

@Var @RT(13)mbRestartMeas @RT(0) @T @F @DT @RT(4)BOOL @RT(0) @T @T @BASIC 0 @F
@F @F
@T
@BEG_Attrib
3 @RT(0) @RT(0) @RT(0)
@END_Attrib
1 0 @F @F @F @F

@Var @RT(14)abSpeedMeasure @RT(0) @T @T @DERIVED 0 @T @T @DT @RT(23)ABAutoIdentSpeedMeasure @RT(0) @T @T @UNKNOWN 0 @F
@F @F
@T
@BEG_Attrib
3 @RT(0) @RT(0) @RT(0)
@END_Attrib
1 0 @F @F @F @F

@Var @RT(13)mrRefVelocity @RT(0) @T @F @DT @RT(4)REAL @RT(0) @T @T @BASIC 0 @F
@F @F
@T
@BEG_Attrib
3 @RT(0) @RT(0) @RT(0)
@END_Attrib
1 0 @F @F @F @F

@Var @RT(13)mrRefPressure @RT(0) @T @F @DT @RT(4)REAL @RT(0) @T @T @BASIC 0 @F
@F @F
@T
@BEG_Attrib
3 @RT(0) @RT(0) @RT(0)
@END_Attrib
1 0 @F @F @F @F

@Var @RT(18)mrMaxLimitPosition @RT(0) @T @F @DT @RT(4)REAL @RT(0) @T @T @BASIC 0 @F
@F @F
@T
@BEG_Attrib
3 @RT(0) @RT(0) @RT(0)
@END_Attrib
1 0 @F @F @F @F

@Var @RT(18)mrMinLimitPosition @RT(0) @T @F @DT @RT(4)REAL @RT(0) @T @T @BASIC 0 @F
@F @F
@T
@BEG_Attrib
3 @RT(0) @RT(0) @RT(0)
@END_Attrib
1 0 @F @F @F @F

@Var @RT(5)dummy @RT(0) @T @F @DT @RT(4)DINT @RT(0) @T @T @BASIC 0 @F
@F @F
@T
@BEG_Attrib
3 @RT(0) @RT(0) @RT(0)
@END_Attrib
1 0 @F @F @F @F

@Var @RT(19)mrMinPositionFactor @RT(0) @T @F @DT @RT(4)REAL @RT(0) @T @T @BASIC 0 @F
@F @F
@T
@BEG_Attrib
3 @RT(3)0.2 @RT(13)20% of stroke @RT(0)
@END_Attrib
1 0 @F @F @F @F

@Var @RT(19)mrMaxPositionFactor @RT(0) @T @F @DT @RT(4)REAL @RT(0) @T @T @BASIC 0 @F
@F @F
@T
@BEG_Attrib
3 @RT(3)0.8 @RT(13)80% of stroke @RT(0)
@END_Attrib
1 0 @F @F @F @F

@Var @RT(13)mrMaxVelocity @RT(0) @T @F @DT @RT(4)REAL @RT(0) @T @T @BASIC 0 @F
@F @F
@T
@BEG_Attrib
3 @RT(0) @RT(0) @RT(0)
@END_Attrib
1 0 @F @F @F @F

@Var @RT(13)mrMaxPressure @RT(0) @T @F @DT @RT(4)REAL @RT(0) @T @T @BASIC 0 @F
@F @F
@T
@BEG_Attrib
3 @RT(0) @RT(0) @RT(0)
@END_Attrib
1 0 @F @F @F @F

@Var @RT(22)mbVelocityLimitReached @RT(0) @T @F @DT @RT(4)BOOL @RT(0) @T @T @BASIC 0 @F
@F @F
@T
@BEG_Attrib
3 @RT(0) @RT(0) @RT(0)
@END_Attrib
1 0 @F @F @F @F

@Var @RT(22)mbPressureLimitReached @RT(0) @T @F @DT @RT(4)BOOL @RT(0) @T @T @BASIC 0 @F
@F @F
@T
@BEG_Attrib
3 @RT(0) @RT(0) @RT(0)
@END_Attrib
1 0 @F @F @F @F

@Var @RT(9)miErrorNo @RT(0) @T @F @DT @RT(3)INT @RT(0) @T @T @BASIC 0 @F
@F @F
@T
@BEG_Attrib
3 @RT(0) @RT(0) @RT(0)
@END_Attrib
1 0 @F @F @F @F

@Var @RT(22)cIdentSpeedMaxSequence @RT(0) @T @F @DT @RT(3)INT @RT(0) @T @T @BASIC 0 @F
@F @F
@T
@BEG_Attrib
3 @RT(3)100 @RT(0) @RT(0)
@END_Attrib
1 0 @F @F @F @F

@Var @RT(22)cIdentSpeedMinSequence @RT(0) @T @F @DT @RT(3)INT @RT(0) @T @T @BASIC 0 @F
@F @F
@T
@BEG_Attrib
3 @RT(3)200 @RT(0) @RT(0)
@END_Attrib
1 0 @F @F @F @F

@Var @RT(22)cIdentSpeedMaxFwdIdent @RT(0) @T @F @DT @RT(3)INT @RT(0) @T @T @BASIC 0 @F
@F @F
@T
@BEG_Attrib
3 @RT(3)101 @RT(0) @RT(0)
@END_Attrib
1 0 @F @F @F @F

@Var @RT(22)cIdentSpeedMinFwdIdent @RT(0) @T @F @DT @RT(3)INT @RT(0) @T @T @BASIC 0 @F
@F @F
@T
@BEG_Attrib
3 @RT(3)201 @RT(0) @RT(0)
@END_Attrib
1 0 @F @F @F @F

@Var @RT(22)cIdentSpeedMaxBwdIdent @RT(0) @T @F @DT @RT(3)INT @RT(0) @T @T @BASIC 0 @F
@F @F
@T
@BEG_Attrib
3 @RT(3)102 @RT(0) @RT(0)
@END_Attrib
1 0 @F @F @F @F

@Var @RT(22)cIdentSpeedMinBwdIdent @RT(0) @T @F @DT @RT(3)INT @RT(0) @T @T @BASIC 0 @F
@F @F
@T
@BEG_Attrib
3 @RT(3)202 @RT(0) @RT(0)
@END_Attrib
1 0 @F @F @F @F

@Var @RT(21)cIdentSpeedMaxBwdInit @RT(0) @T @F @DT @RT(3)INT @RT(0) @T @T @BASIC 0 @F
@F @F
@T
@BEG_Attrib
3 @RT(3)103 @RT(0) @RT(0)
@END_Attrib
1 0 @F @F @F @F

@Var @RT(21)cIdentSpeedMinBwdInit @RT(0) @T @F @DT @RT(3)INT @RT(0) @T @T @BASIC 0 @F
@F @F
@T
@BEG_Attrib
3 @RT(3)203 @RT(0) @RT(0)
@END_Attrib
1 0 @F @F @F @F

@Var @RT(21)cIdentSpeedMaxFwdInit @RT(0) @T @F @DT @RT(3)INT @RT(0) @T @T @BASIC 0 @F
@F @F
@T
@BEG_Attrib
3 @RT(3)104 @RT(0) @RT(0)
@END_Attrib
1 0 @F @F @F @F

@Var @RT(21)cIdentSpeedMinFwdInit @RT(0) @T @F @DT @RT(3)INT @RT(0) @T @T @BASIC 0 @F
@F @F
@T
@BEG_Attrib
3 @RT(3)204 @RT(0) @RT(0)
@END_Attrib
1 0 @F @F @F @F

@Var @RT(22)cIdentSpeedMaxFwdStart @RT(0) @T @F @DT @RT(3)INT @RT(0) @T @T @BASIC 0 @F
@F @F
@T
@BEG_Attrib
3 @RT(3)105 @RT(0) @RT(0)
@END_Attrib
1 0 @F @F @F @F

@Var @RT(22)cIdentSpeedMinFwdStart @RT(0) @T @F @DT @RT(3)INT @RT(0) @T @T @BASIC 0 @F
@F @F
@T
@BEG_Attrib
3 @RT(3)205 @RT(0) @RT(0)
@END_Attrib
1 0 @F @F @F @F

@Var @RT(22)cIdentSpeedMaxBwdStart @RT(0) @T @F @DT @RT(3)INT @RT(0) @T @T @BASIC 0 @F
@F @F
@T
@BEG_Attrib
3 @RT(3)106 @RT(0) @RT(0)
@END_Attrib
1 0 @F @F @F @F

@Var @RT(22)cIdentSpeedMinBwdStart @RT(0) @T @F @DT @RT(3)INT @RT(0) @T @T @BASIC 0 @F
@F @F
@T
@BEG_Attrib
3 @RT(3)206 @RT(0) @RT(0)
@END_Attrib
1 0 @F @F @F @F

@Var @RT(17)cIdentSpeedMaxEnd @RT(0) @T @F @DT @RT(3)INT @RT(0) @T @T @BASIC 0 @F
@F @F
@T
@BEG_Attrib
3 @RT(3)107 @RT(0) @RT(0)
@END_Attrib
1 0 @F @F @F @F

@Var @RT(17)cIdentSpeedMinEnd @RT(0) @T @F @DT @RT(3)INT @RT(0) @T @T @BASIC 0 @F
@F @F
@T
@BEG_Attrib
3 @RT(3)207 @RT(0) @RT(0)
@END_Attrib
1 0 @F @F @F @F

@Var @RT(17)mrBwdStopPosition @RT(0) @T @F @DT @RT(4)REAL @RT(0) @T @T @BASIC 0 @F
@F @F
@T
@BEG_Attrib
3 @RT(4)0.05 @RT(0) @RT(0)
@END_Attrib
1 0 @F @F @F @F

@Var @RT(14)mprActPressure @RT(0) @T @T @REFTO 0 @T @DT @RT(4)REAL @RT(0) @T @T @BASIC 0 @F
@F @F
@T
@BEG_Attrib
3 @RT(0) @RT(0) @RT(0)
@END_Attrib
1 0 @F @F @F @F

@Var @RT(21)mbprActPressureLinked @RT(0) @T @F @DT @RT(4)BOOL @RT(0) @T @T @BASIC 0 @F
@F @F
@T
@BEG_Attrib
3 @RT(0) @RT(0) @RT(0)
@END_Attrib
1 0 @F @F @F @F

@Var @RT(10)PU_Task_13 @RT(0) @T @F @DT @RT(4)TASK @RT(0) @T @T @BASIC 0 @F
@F @F
@T
@BEG_Attrib
3 @RT(0) @RT(0) @RT(0)
@END_Attrib
1 7 @F @F @F @F

@Var @RT(12)sv_DataState @RT(0) @T @T @DERIVED 0 @T @T @DT @RT(11)tnDataState @RT(0) @T @T @UNKNOWN 0 @F
@F @F
@T
@BEG_Attrib
3 @RT(0) @RT(0) @RT(0)
@END_Attrib
1 8 @F @F @F @F

@END_Dcl

@END_Export

@BEG_Body

28

@BEG_Export

@BEG_Algo
@PROCESS_ALGORITHM @RT(6)paInit @STRUCTURED_TEXT
@RT(0) @RT(0) @RT(7)TaskMid @T @F
@END_Algo

@BEG_Dcl
@RT(16)DclTreeContainer
7
@Var @RT(1)j @RT(0) @T @F @DT @RT(4)DINT @RT(0) @T @T @BASIC 0 @F
@F @F
@T
@BEG_Attrib
3 @RT(0) @RT(0) @RT(0)
@END_Attrib
1 4 @F @F @F @F

@Var @RT(1)k @RT(0) @T @F @DT @RT(4)DINT @RT(0) @T @T @BASIC 0 @F
@F @F
@T
@BEG_Attrib
3 @RT(0) @RT(0) @RT(0)
@END_Attrib
1 4 @F @F @F @F

@Var @RT(1)i @RT(0) @T @F @DT @RT(4)DINT @RT(0) @T @T @BASIC 0 @F
@F @F
@T
@BEG_Attrib
3 @RT(0) @RT(0) @RT(0)
@END_Attrib
1 0 @F @F @F @F

@Var @RT(6)Status @RT(0) @T @T @DERIVED 0 @T @T @DT @RT(11)KSYS_Status @RT(0) @T @T @UNKNOWN 0 @F
@F @F
@T
@BEG_Attrib
3 @RT(0) @RT(0) @RT(0)
@END_Attrib
1 0 @F @F @F @F

@Var @RT(10)rpPosition @RT(0) @T @T @REFTO 0 @T @DT @RT(4)REAL @RT(0) @T @T @BASIC 0 @F
@F @F
@T
@BEG_Attrib
3 @RT(0) @RT(0) @RT(0)
@END_Attrib
1 0 @F @F @F @F

@Var @RT(4)tmpM @RT(0) @T @T @DERIVED 0 @T @T @DT @RT(20)tpIdentSpeedMovement @RT(0) @T @T @UNKNOWN 0 @F
@F @F
@T
@BEG_Attrib
3 @RT(0) @RT(0) @RT(0)
@END_Attrib
1 0 @F @F @F @F

@Var @RT(7)pOption @RT(0) @T @T @REFTO 0 @F @DERIVED 0 @T @T @DT @RT(9)tOptionId @RT(0) @T @T @UNKNOWN 0 @F
@F @F
@T
@BEG_Attrib
3 @RT(0) @RT(0) @RT(0)
@END_Attrib
1 0 @F @F @F @F

@END_Dcl

@END_Export

@BEG_Export

@BEG_Algo
@POSTUPDATE_ALGORITHM @RT(13)pAlarmPending @STRUCTURED_TEXT
@RT(0) @RT(17)sv_iPendingAlarms @RT(9)PU_Task_7 @F @F
@END_Algo

@BEG_Dcl
@RT(16)DclTreeContainer
1
@Var @RT(20)fbTracePendingAlarms @RT(0) @T @T @DERIVED 0 @T @T @DT @RT(20)FBTracePendingAlarms @RT(0) @T @T @UNKNOWN 0 @F
@F @F
@T
@BEG_Attrib
3 @RT(0) @RT(0) @RT(0)
@END_Attrib
1 0 @F @F @F @F

@END_Dcl

@END_Export

@BEG_Export

@BEG_Algo
@ALGORITHM @RT(8)aMeasure @STRUCTURED_TEXT
@RT(0) @RT(0) @RT(0) @F @F
@END_Algo

@BEG_Dcl
@RT(16)DclTreeContainer
1
@Var @RT(12)rActPressure @RT(0) @T @F @DT @RT(4)REAL @RT(0) @T @T @BASIC 0 @F
@F @F
@T
@BEG_Attrib
3 @RT(0) @RT(0) @RT(0)
@END_Attrib
1 0 @F @F @F @F

@END_Dcl

@END_Export

@BEG_Export

@BEG_Algo
@PROCESS_ALGORITHM @RT(13)paMeasureFast @STRUCTURED_TEXT
@RT(0) @RT(0) @RT(10)TaskInject @F @F
@END_Algo

@BEG_Dcl
@RT(16)DclTreeContainer
0
@END_Dcl

@END_Export

@BEG_Export

@BEG_Algo
@PROCESS_ALGORITHM @RT(12)paMeasureMid @STRUCTURED_TEXT
@RT(0) @RT(0) @RT(10)TaskAnalog @F @F
@END_Algo

@BEG_Dcl
@RT(16)DclTreeContainer
0
@END_Dcl

@END_Export

@BEG_Export

@BEG_Algo
@ALGORITHM @RT(17)aStartMeasurement @STRUCTURED_TEXT
@RT(0) @RT(0) @RT(0) @F @F
@END_Algo

@BEG_Dcl
@RT(16)DclTreeContainer
0
@END_Dcl

@END_Export

@BEG_Export

@BEG_Algo
@ALGORITHM @RT(16)aStopMeasurement @STRUCTURED_TEXT
@RT(0) @RT(0) @RT(0) @F @F
@END_Algo

@BEG_Dcl
@RT(16)DclTreeContainer
0
@END_Dcl

@END_Export

@BEG_Export

@BEG_Algo
@ALGORITHM @RT(9)aWriteLog @STRUCTURED_TEXT
@RT(0) @RT(0) @RT(0) @F @F
@END_Algo

@BEG_Dcl
@RT(16)DclTreeContainer
3
@Var @RT(9)sFileName @RT(0) @T @F @DT @RT(11)STRING(255) @RT(0) @T @T @STRING 0 @F @RT(3)255 @F
@F @F
@T
@BEG_Attrib
3 @RT(0) @RT(18)file name movement @RT(0)
@END_Attrib
1 1 @F @F @F @F

@Var @RT(12)iFileCounter @RT(0) @T @F @DT @RT(5)UDINT @RT(0) @T @T @BASIC 0 @F
@F @F
@T
@BEG_Attrib
3 @RT(0) @RT(24)actual ident cycle index @RT(0)
@END_Attrib
1 1 @F @F @F @F

@Var @RT(12)bDeleteFiles @RT(0) @T @F @DT @RT(4)BOOL @RT(0) @T @T @BASIC 0 @F
@F @F
@T
@BEG_Attrib
3 @RT(0) @RT(16)delete old files @RT(0)
@END_Attrib
1 1 @F @F @F @F

@END_Dcl

@END_Export

@BEG_Export

@BEG_Algo
@PROCESS_ALGORITHM @RT(10)paWriteLog @STRUCTURED_TEXT
@RT(0) @RT(0) @RT(8)TaskSlow @F @F
@END_Algo

@BEG_Dcl
@RT(16)DclTreeContainer
0
@END_Dcl

@END_Export

@BEG_Export

@BEG_Algo
@ALGORITHM @RT(17)aStartMovementFwd @STRUCTURED_TEXT
@RT(0) @RT(0) @RT(0) @F @F
@END_Algo

@BEG_Dcl
@RT(16)DclTreeContainer
0
@END_Dcl

@END_Export

@BEG_Export

@BEG_Algo
@ALGORITHM @RT(17)aStartMovementBwd @STRUCTURED_TEXT
@RT(0) @RT(0) @RT(0) @F @F
@END_Algo

@BEG_Dcl
@RT(16)DclTreeContainer
0
@END_Dcl

@END_Export

@BEG_Export

@BEG_Algo
@ALGORITHM @RT(16)aStopMovementFwd @STRUCTURED_TEXT
@RT(0) @RT(0) @RT(0) @F @F
@END_Algo

@BEG_Dcl
@RT(16)DclTreeContainer
0
@END_Dcl

@END_Export

@BEG_Export

@BEG_Algo
@ALGORITHM @RT(16)aStopMovementBwd @STRUCTURED_TEXT
@RT(0) @RT(0) @RT(0) @F @F
@END_Algo

@BEG_Dcl
@RT(16)DclTreeContainer
0
@END_Dcl

@END_Export

@BEG_Export

@BEG_Algo
@ALGORITHM @RT(18)aStopMovementError @STRUCTURED_TEXT
@RT(0) @RT(0) @RT(0) @F @F
@END_Algo

@BEG_Dcl
@RT(16)DclTreeContainer
1
@Var @RT(13)sMovementName @RT(0) @T @F @DT @RT(11)STRING(255) @RT(0) @T @T @STRING 0 @F @RT(3)255 @F
@F @F
@T
@BEG_Attrib
3 @RT(0) @RT(20)Movement information @RT(0)
@END_Attrib
1 1 @F @F @F @F

@END_Dcl

@END_Export

@BEG_Export

@BEG_Algo
@ALGORITHM @RT(19)aCalcMaxSpeedOutput @STRUCTURED_TEXT
@RT(0) @RT(0) @RT(0) @F @F
@END_Algo

@BEG_Dcl
@RT(16)DclTreeContainer
12
@Var @RT(14)rMaxSpeedLimit @RT(0) @T @F @DT @RT(4)REAL @RT(0) @T @T @BASIC 0 @F
@F @F
@T
@BEG_Attrib
3 @RT(0) @RT(36)Maximum speed limit of actual device @RT(0)
@END_Attrib
1 1 @F @F @F @F

@Var @RT(14)rActSpeedLimit @RT(0) @T @F @DT @RT(4)REAL @RT(0) @T @T @BASIC 0 @F
@F @F
@T
@BEG_Attrib
3 @RT(0) @RT(35)Actual speed limit of actual device @RT(0)
@END_Attrib
1 1 @F @F @F @F

@Var @RT(12)rActMaxSpeed @RT(0) @T @F @DT @RT(4)REAL @RT(0) @T @T @BASIC 0 @F
@F @F
@T
@BEG_Attrib
3 @RT(0) @RT(22)Maximum measured speed @RT(0)
@END_Attrib
1 1 @F @F @F @F

@Var @RT(17)bPresLimitReached @RT(0) @T @F @DT @RT(4)BOOL @RT(0) @T @T @BASIC 0 @F
@F @F
@T
@BEG_Attrib
3 @RT(0) @RT(38)Pressure limit reached during movement @RT(0)
@END_Attrib
1 1 @F @F @F @F

@Var @RT(16)bUsePressureMode @RT(0) @T @F @DT @RT(4)BOOL @RT(0) @T @T @BASIC 0 @F
@F @F
@T
@BEG_Attrib
3 @RT(0) @RT(80)Use pressure to check maimum speed limit reached. Otherwise use actual  velocity @RT(0)
@END_Attrib
1 1 @F @F @F @F

@Var @RT(12)bMaxDetected @RT(0) @T @F @DT @RT(4)BOOL @RT(0) @T @T @BASIC 0 @F
@F @F
@T
@BEG_Attrib
3 @RT(0) @RT(20)Speed limit detected @RT(0)
@END_Attrib
1 3 @F @F @F @F

@Var @RT(9)rRefSpeed @RT(0) @T @F @DT @RT(4)REAL @RT(0) @T @T @BASIC 0 @F
@F @F
@T
@BEG_Attrib
3 @RT(0) @RT(24)Speed limit for next try @RT(0)
@END_Attrib
1 3 @F @F @F @F

@Var @RT(9)rMaxSpeed @RT(0) @T @F @DT @RT(4)REAL @RT(0) @T @T @BASIC 0 @F
@F @F
@T
@BEG_Attrib
3 @RT(0) @RT(20)Identified max speed @RT(0)
@END_Attrib
1 3 @F @F @F @F

@Var @RT(19)rSpeedReachedFactor @RT(0) @T @F @DT @RT(4)REAL @RT(0) @T @T @BASIC 0 @F
@F @F
@T
@BEG_Attrib
3 @RT(4)0.95 @RT(0) @RT(0)
@END_Attrib
1 0 @F @F @F @F

@Var @RT(12)rMaxActSpeed @RT(0) @T @F @DT @RT(4)REAL @RT(0) @T @T @BASIC 0 @F
@F @F
@T
@BEG_Attrib
3 @RT(0) @RT(0) @RT(0)
@END_Attrib
1 0 @F @F @F @F

@Var @RT(12)rMinActSpeed @RT(0) @T @F @DT @RT(4)REAL @RT(0) @T @T @BASIC 0 @F
@F @F
@T
@BEG_Attrib
3 @RT(3)0.0 @RT(0) @RT(0)
@END_Attrib
1 0 @F @F @F @F

@Var @RT(19)rMinSpeedDifference @RT(0) @T @F @DT @RT(4)REAL @RT(0) @T @T @BASIC 0 @F
@F @F
@T
@BEG_Attrib
3 @RT(4)0.05 @RT(0) @RT(0)
@END_Attrib
1 0 @F @F @F @F

@END_Dcl

@END_Export

@BEG_Export

@BEG_Algo
@EVENT_ALGORITHM @RT(15)evaRedoMaxEvent @STRUCTURED_TEXT
@RT(0) @RT(24)evRedoIdentMaxSpeedStart @RT(9)EV_Task_7 @F @F
@END_Algo

@BEG_Dcl
@RT(16)DclTreeContainer
1
@Var @RT(20)evRedoIdentEventData @RT(0) @T @T @DERIVED 0 @T @T @DT @RT(26)tevRedoIdentSpeedEventData @RT(0) @T @T @UNKNOWN 0 @F
@F @F
@T
@BEG_Attrib
3 @RT(0) @RT(44)Event data to start max speed identification @RT(0)
@END_Attrib
1 1 @F @F @F @F

@END_Dcl

@END_Export

@BEG_Export

@BEG_Algo
@PROCESS_ALGORITHM @RT(9)paRedoMax @STRUCTURED_TEXT
@RT(0) @RT(0) @RT(7)TaskMid @F @F
@END_Algo

@BEG_Dcl
@RT(16)DclTreeContainer
2
@Var @RT(1)i @RT(0) @T @F @DT @RT(4)DINT @RT(0) @T @T @BASIC 0 @F
@F @F
@T
@BEG_Attrib
3 @RT(0) @RT(0) @RT(0)
@END_Attrib
1 4 @F @F @F @F

@Var @RT(12)bIdentActive @RT(0) @T @F @DT @RT(4)BOOL @RT(0) @T @T @BASIC 0 @F
@F @F
@T
@BEG_Attrib
3 @RT(0) @RT(0) @RT(0)
@END_Attrib
1 4 @F @F @F @F

@END_Dcl

@END_Export

@BEG_Export

@BEG_Algo
@PROCESS_ALGORITHM @RT(19)paMaxSingleMovement @SEQUENTIAL_FLOW_CHART
@RT(0) @RT(0) @RT(7)TaskMid @F @F
@END_Algo

@BEG_Dcl
@RT(16)DclTreeContainer
28
@Var @RT(12)bMoveBwdDone @RT(0) @T @F @DT @RT(4)BOOL @RT(0) @T @T @BASIC 0 @F
@F @F
@T
@BEG_Attrib
3 @RT(5)FALSE @RT(0) @RT(0)
@END_Attrib
1 0 @F @F @F @F

@Var @RT(12)bMoveFwdDone @RT(0) @T @F @DT @RT(4)BOOL @RT(0) @T @T @BASIC 0 @F
@F @F
@T
@BEG_Attrib
3 @RT(5)FALSE @RT(0) @RT(0)
@END_Attrib
1 0 @F @F @F @F

@Var @RT(14)bMoveIdentDone @RT(0) @T @F @DT @RT(4)BOOL @RT(0) @T @T @BASIC 0 @F
@F @F
@T
@BEG_Attrib
3 @RT(5)FALSE @RT(0) @RT(0)
@END_Attrib
1 0 @F @F @F @F

@Var @RT(9)sFileName @RT(0) @T @F @DT @RT(11)STRING(255) @RT(0) @T @T @STRING 0 @F @RT(3)255 @F
@F @F
@T
@BEG_Attrib
3 @RT(0) @RT(0) @RT(0)
@END_Attrib
1 0 @F @F @F @F

@Var @RT(12)iFileCounter @RT(0) @T @F @DT @RT(5)UDINT @RT(0) @T @T @BASIC 0 @F
@F @F
@T
@BEG_Attrib
3 @RT(1)1 @RT(0) @RT(0)
@END_Attrib
1 0 @F @F @F @F

@Var @RT(8)ConstVis @RT(0) @T @T @DERIVED 0 @T @T @DT @RT(8)tsVelPre @RT(0) @T @T @UNKNOWN 0 @F
@F @F
@T
@BEG_Attrib
3 @RT(0) @RT(41)const output for ejector forward movement @RT(0)
@END_Attrib
1 0 @F @F @F @F

@Var @RT(11)ConstVisFwd @RT(0) @T @T @DERIVED 0 @T @T @DT @RT(8)tsVelPre @RT(0) @T @T @UNKNOWN 0 @F
@F @F
@T
@BEG_Attrib
3 @RT(0) @RT(41)const output for ejector forward movement @RT(0)
@END_Attrib
1 0 @F @F @F @F

@Var @RT(11)ConstVisBwd @RT(0) @T @T @DERIVED 0 @T @T @DT @RT(8)tsVelPre @RT(0) @T @T @UNKNOWN 0 @F
@F @F
@T
@BEG_Attrib
3 @RT(0) @RT(41)const output for ejector forward movement @RT(0)
@END_Attrib
1 0 @F @F @F @F

@Var @RT(12)bMaxFwdRetry @RT(0) @T @F @DT @RT(4)BOOL @RT(0) @T @T @BASIC 0 @F
@F @F
@T
@BEG_Attrib
3 @RT(0) @RT(0) @RT(0)
@END_Attrib
1 0 @F @F @F @F

@Var @RT(12)bMaxBwdRetry @RT(0) @T @F @DT @RT(4)BOOL @RT(0) @T @T @BASIC 0 @F
@F @F
@T
@BEG_Attrib
3 @RT(0) @RT(0) @RT(0)
@END_Attrib
1 0 @F @F @F @F

@Var @RT(15)bMaxFwdDetected @RT(0) @T @F @DT @RT(4)BOOL @RT(0) @T @T @BASIC 0 @F
@F @F
@T
@BEG_Attrib
3 @RT(0) @RT(0) @RT(0)
@END_Attrib
1 0 @F @F @F @F

@Var @RT(15)bMaxBwdDetected @RT(0) @T @F @DT @RT(4)BOOL @RT(0) @T @T @BASIC 0 @F
@F @F
@T
@BEG_Attrib
3 @RT(0) @RT(0) @RT(0)
@END_Attrib
1 0 @F @F @F @F

@Var @RT(9)sMoveName @RT(0) @T @F @DT @RT(10)STRING(32) @RT(0) @T @T @STRING 0 @F @RT(2)32 @F
@F @F
@T
@BEG_Attrib
3 @RT(0) @RT(0) @RT(0)
@END_Attrib
1 0 @F @F @F @F

@Var @RT(17)rMaxPressureLimit @RT(0) @T @F @DT @RT(4)REAL @RT(0) @T @T @BASIC 0 @F
@F @F
@T
@BEG_Attrib
3 @RT(0) @RT(0) @RT(0)
@END_Attrib
1 0 @F @F @F @F

@Var @RT(14)rRefSpeedLimit @RT(0) @T @F @DT @RT(4)REAL @RT(0) @T @T @BASIC 0 @F
@F @F
@T
@BEG_Attrib
3 @RT(0) @RT(0) @RT(0)
@END_Attrib
1 0 @F @F @F @F

@Var @RT(14)rSpeedLimitFwd @RT(0) @T @F @DT @RT(4)REAL @RT(0) @T @T @BASIC 0 @F
@F @F
@T
@BEG_Attrib
3 @RT(0) @RT(0) @RT(0)
@END_Attrib
1 0 @F @F @F @F

@Var @RT(14)rSpeedLimitBwd @RT(0) @T @F @DT @RT(4)REAL @RT(0) @T @T @BASIC 0 @F
@F @F
@T
@BEG_Attrib
3 @RT(0) @RT(0) @RT(0)
@END_Attrib
1 0 @F @F @F @F

@Var @RT(20)rMaxRefPressureLimit @RT(0) @T @F @DT @RT(4)REAL @RT(0) @T @T @BASIC 0 @F
@F @F
@T
@BEG_Attrib
3 @RT(0) @RT(0) @RT(0)
@END_Attrib
1 0 @F @F @F @F

@Var @RT(16)sWriteSpeedLimit @RT(0) @T @F @DT @RT(11)STRING(255) @RT(0) @T @T @STRING 0 @F @RT(3)255 @F
@F @F
@T
@BEG_Attrib
3 @RT(0) @RT(0) @RT(0)
@END_Attrib
1 0 @F @F @F @F

@Var @RT(18)rVelocitSizeFactor @RT(0) @T @F @DT @RT(4)REAL @RT(0) @T @T @BASIC 0 @F
@F @F
@T
@BEG_Attrib
3 @RT(3)1.0 @RT(0) @RT(0)
@END_Attrib
1 0 @F @F @F @F

@Var @RT(12)rStartFactor @RT(0) @T @F @DT @RT(4)REAL @RT(0) @T @T @BASIC 0 @F
@F @F
@T
@BEG_Attrib
3 @RT(3)0.1 @RT(0) @RT(0)
@END_Attrib
1 0 @F @F @F @F

@Var @RT(12)rMinStopRamp @RT(0) @T @F @DT @RT(4)REAL @RT(0) @T @T @BASIC 0 @F
@F @F
@T
@BEG_Attrib
3 @RT(3)1.0 @RT(0) @RT(0)
@END_Attrib
1 0 @F @F @F @F

@Var @RT(16)rMinStrokeFactor @RT(0) @T @F @DT @RT(4)REAL @RT(0) @T @T @BASIC 0 @F
@F @F
@T
@BEG_Attrib
3 @RT(3)0.5 @RT(0) @RT(0)
@END_Attrib
1 0 @F @F @F @F

@Var @RT(22)bDelayTimeOffFwdLinked @RT(0) @T @F @DT @RT(4)BOOL @RT(0) @T @T @BASIC 0 @F
@F @F
@T
@BEG_Attrib
3 @RT(0) @RT(0) @RT(0)
@END_Attrib
1 0 @F @F @F @F

@Var @RT(22)bDelayTimeOffBwdLinked @RT(0) @T @F @DT @RT(4)BOOL @RT(0) @T @T @BASIC 0 @F
@F @F
@T
@BEG_Attrib
3 @RT(0) @RT(0) @RT(0)
@END_Attrib
1 0 @F @F @F @F

@Var @RT(16)dDelayTimeOffFwd @RT(0) @T @F @DT @RT(4)TIME @RT(0) @T @T @BASIC 0 @F
@F @F
@T
@BEG_Attrib
3 @RT(0) @RT(0) @RT(0)
@END_Attrib
1 0 @F @F @F @F

@Var @RT(16)dDelayTimeOffBwd @RT(0) @T @F @DT @RT(4)TIME @RT(0) @T @T @BASIC 0 @F
@F @F
@T
@BEG_Attrib
3 @RT(0) @RT(0) @RT(0)
@END_Attrib
1 0 @F @F @F @F

@Var @RT(16)dMinDelayTimeOff @RT(0) @T @F @DT @RT(4)TIME @RT(0) @T @T @BASIC 0 @F
@F @F
@T
@BEG_Attrib
3 @RT(6)T#25ms @RT(0) @RT(0)
@END_Attrib
1 0 @F @F @F @F

@END_Dcl

@END_Export

@BEG_Export

@BEG_Algo
@POSTUPDATE_ALGORITHM @RT(17)pMaxCommandListen @STRUCTURED_TEXT
@RT(0) @RT(72)sv_GlobalIdentMaxSpeedStatus.Command,sv_GlobalIdentMaxSpeedStatus.bStart @RT(9)PU_Task_7 @F @F
@END_Algo

@BEG_Dcl
@RT(16)DclTreeContainer
1
@Var @RT(1)i @RT(0) @T @F @DT @RT(4)DINT @RT(0) @T @T @BASIC 0 @F
@F @F
@T
@BEG_Attrib
3 @RT(0) @RT(0) @RT(0)
@END_Attrib
1 4 @F @F @F @F

@END_Dcl

@END_Export

@BEG_Export

@BEG_Algo
@PROCESS_ALGORITHM @RT(18)paMaxCalibSequence @SEQUENTIAL_FLOW_CHART
@RT(0) @RT(0) @RT(7)TaskMid @F @F
@END_Algo

@BEG_Dcl
@RT(16)DclTreeContainer
6
@Var @RT(1)j @RT(0) @T @F @DT @RT(4)DINT @RT(0) @T @T @BASIC 0 @F
@F @F
@T
@BEG_Attrib
3 @RT(0) @RT(0) @RT(0)
@END_Attrib
1 4 @F @F @F @F

@Var @RT(1)i @RT(0) @T @F @DT @RT(4)DINT @RT(0) @T @T @BASIC 0 @F
@F @F
@T
@BEG_Attrib
3 @RT(0) @RT(0) @RT(0)
@END_Attrib
1 4 @F @F @F @F

@Var @RT(12)tmpMovements @RT(0) @T @T @DERIVED 0 @T @T @DT @RT(21)tyIdentSpeedMovements @RT(0) @T @T @UNKNOWN 0 @F
@F @F
@T
@BEG_Attrib
3 @RT(0) @RT(0) @RT(0)
@END_Attrib
1 0 @F @F @F @F

@Var @RT(13)iMaxMovements @RT(0) @T @F @DT @RT(4)DINT @RT(0) @T @T @BASIC 0 @F
@F @F
@T
@BEG_Attrib
3 @RT(0) @RT(0) @RT(0)
@END_Attrib
1 0 @F @F @F @F

@Var @RT(4)tmpM @RT(0) @T @T @DERIVED 0 @T @T @DT @RT(20)tpIdentSpeedMovement @RT(0) @T @T @UNKNOWN 0 @F
@F @F
@T
@BEG_Attrib
3 @RT(0) @RT(0) @RT(0)
@END_Attrib
1 0 @F @F @F @F

@Var @RT(11)ConstBwdVis @RT(0) @T @T @DERIVED 0 @T @T @DT @RT(8)tsVelPre @RT(0) @T @T @UNKNOWN 0 @F
@F @F
@T
@BEG_Attrib
3 @RT(0) @RT(0) @RT(0)
@END_Attrib
1 0 @F @F @F @F

@END_Dcl

@END_Export

@BEG_Export

@BEG_Algo
@ALGORITHM @RT(6)aRound @STRUCTURED_TEXT
@RT(0) @RT(0) @RT(0) @F @F
@END_Algo

@BEG_Dcl
@RT(16)DclTreeContainer
4
@Var @RT(10)rActNumber @RT(0) @T @F @DT @RT(4)REAL @RT(0) @T @T @BASIC 0 @F
@F @F
@T
@BEG_Attrib
3 @RT(0) @RT(0) @RT(0)
@END_Attrib
1 1 @F @F @F @F

@Var @RT(5)rStep @RT(0) @T @F @DT @RT(4)REAL @RT(0) @T @T @BASIC 0 @F
@F @F
@T
@BEG_Attrib
3 @RT(0) @RT(0) @RT(0)
@END_Attrib
1 1 @F @F @F @F

@Var @RT(14)rRoundedNumber @RT(0) @T @F @DT @RT(4)REAL @RT(0) @T @T @BASIC 0 @F
@F @F
@T
@BEG_Attrib
3 @RT(0) @RT(0) @RT(0)
@END_Attrib
1 3 @F @F @F @F

@Var @RT(10)rRealValue @RT(0) @T @F @DT @RT(4)REAL @RT(0) @T @T @BASIC 0 @F
@F @F
@T
@BEG_Attrib
3 @RT(0) @RT(0) @RT(0)
@END_Attrib
1 0 @F @F @F @F

@END_Dcl

@END_Export

@BEG_Export

@BEG_Algo
@ALGORITHM @RT(19)aCalcMinSpeedOutput @STRUCTURED_TEXT
@RT(0) @RT(0) @RT(0) @F @F
@END_Algo

@BEG_Dcl
@RT(16)DclTreeContainer
12
@Var @RT(6)bStart @RT(0) @T @F @DT @RT(4)BOOL @RT(0) @T @T @BASIC 0 @F
@F @F
@T
@BEG_Attrib
3 @RT(0) @RT(58)Restart calculation of reference for min speed calibration @RT(0)
@END_Attrib
1 1 @F @F @F @F

@Var @RT(14)rMaxSpeedLimit @RT(0) @T @F @DT @RT(4)REAL @RT(0) @T @T @BASIC 0 @F
@F @F
@T
@BEG_Attrib
3 @RT(0) @RT(36)Maximum speed limit of actual device @RT(0)
@END_Attrib
1 1 @F @F @F @F

@Var @RT(12)rActRefSpeed @RT(0) @T @F @DT @RT(4)REAL @RT(0) @T @T @BASIC 0 @F
@F @F
@T
@BEG_Attrib
3 @RT(0) @RT(35)Actual speed limit of actual device @RT(0)
@END_Attrib
1 1 @F @F @F @F

@Var @RT(12)rActMinSpeed @RT(0) @T @F @DT @RT(4)REAL @RT(0) @T @T @BASIC 0 @F
@F @F
@T
@BEG_Attrib
3 @RT(0) @RT(22)Minimum measured speed @RT(0)
@END_Attrib
1 1 @F @F @F @F

@Var @RT(9)bUnstable @RT(0) @T @F @DT @RT(4)BOOL @RT(0) @T @T @BASIC 0 @F
@F @F
@T
@BEG_Attrib
3 @RT(0) @RT(23)Measured speed unstable @RT(0)
@END_Attrib
1 1 @F @F @F @F

@Var @RT(8)bTimeOut @RT(0) @T @F @DT @RT(4)BOOL @RT(0) @T @T @BASIC 0 @F
@F @F
@T
@BEG_Attrib
3 @RT(0) @RT(41)Timeout during movement aof actual device @RT(0)
@END_Attrib
1 1 @F @F @F @F

@Var @RT(12)bMinDetected @RT(0) @T @F @DT @RT(4)BOOL @RT(0) @T @T @BASIC 0 @F
@F @F
@T
@BEG_Attrib
3 @RT(0) @RT(20)Speed limit detected @RT(0)
@END_Attrib
1 3 @F @F @F @F

@Var @RT(9)rRefSpeed @RT(0) @T @F @DT @RT(4)REAL @RT(0) @T @T @BASIC 0 @F
@F @F
@T
@BEG_Attrib
3 @RT(0) @RT(24)Speed limit for next try @RT(0)
@END_Attrib
1 3 @F @F @F @F

@Var @RT(9)rMinSpeed @RT(0) @T @F @DT @RT(4)REAL @RT(0) @T @T @BASIC 0 @F
@F @F
@T
@BEG_Attrib
3 @RT(0) @RT(21)Identified min output @RT(0)
@END_Attrib
1 3 @F @F @F @F

@Var @RT(12)rMaxRefSpeed @RT(0) @T @F @DT @RT(4)REAL @RT(0) @T @T @BASIC 0 @F
@F @F
@T
@BEG_Attrib
3 @RT(0) @RT(0) @RT(0)
@END_Attrib
1 0 @F @F @F @F

@Var @RT(12)rMinRefSpeed @RT(0) @T @F @DT @RT(4)REAL @RT(0) @T @T @BASIC 0 @F
@F @F
@T
@BEG_Attrib
3 @RT(3)0.0 @RT(0) @RT(0)
@END_Attrib
1 0 @F @F @F @F

@Var @RT(19)rMFactorMaxMinLimit @RT(0) @T @F @DT @RT(4)REAL @RT(0) @T @T @BASIC 0 @F
@F @F
@T
@BEG_Attrib
3 @RT(3)0.2 @RT(0) @RT(0)
@END_Attrib
1 0 @F @F @F @F

@END_Dcl

@END_Export

@BEG_Export

@BEG_Algo
@PROCESS_ALGORITHM @RT(9)paRedoMin @STRUCTURED_TEXT
@RT(0) @RT(0) @RT(7)TaskMid @F @F
@END_Algo

@BEG_Dcl
@RT(16)DclTreeContainer
2
@Var @RT(1)i @RT(0) @T @F @DT @RT(4)DINT @RT(0) @T @T @BASIC 0 @F
@F @F
@T
@BEG_Attrib
3 @RT(0) @RT(0) @RT(0)
@END_Attrib
1 4 @F @F @F @F

@Var @RT(12)bIdentActive @RT(0) @T @F @DT @RT(4)BOOL @RT(0) @T @T @BASIC 0 @F
@F @F
@T
@BEG_Attrib
3 @RT(0) @RT(0) @RT(0)
@END_Attrib
1 4 @F @F @F @F

@END_Dcl

@END_Export

@BEG_Export

@BEG_Algo
@EVENT_ALGORITHM @RT(15)evaRedoMinEvent @STRUCTURED_TEXT
@RT(0) @RT(24)evRedoIdentMinSpeedStart @RT(9)EV_Task_7 @F @F
@END_Algo

@BEG_Dcl
@RT(16)DclTreeContainer
1
@Var @RT(20)evRedoIdentEventData @RT(0) @T @T @DERIVED 0 @T @T @DT @RT(26)tevRedoIdentSpeedEventData @RT(0) @T @T @UNKNOWN 0 @F
@F @F
@T
@BEG_Attrib
3 @RT(0) @RT(44)Event data to start min speed identification @RT(0)
@END_Attrib
1 1 @F @F @F @F

@END_Dcl

@END_Export

@BEG_Export

@BEG_Algo
@PROCESS_ALGORITHM @RT(19)paMinSingleMovement @SEQUENTIAL_FLOW_CHART
@RT(0) @RT(0) @RT(7)TaskMid @F @F
@END_Algo

@BEG_Dcl
@RT(16)DclTreeContainer
39
@Var @RT(12)bMoveBwdDone @RT(0) @T @F @DT @RT(4)BOOL @RT(0) @T @T @BASIC 0 @F
@F @F
@T
@BEG_Attrib
3 @RT(5)FALSE @RT(0) @RT(0)
@END_Attrib
1 0 @F @F @F @F

@Var @RT(12)bMoveFwdDone @RT(0) @T @F @DT @RT(4)BOOL @RT(0) @T @T @BASIC 0 @F
@F @F
@T
@BEG_Attrib
3 @RT(5)FALSE @RT(0) @RT(0)
@END_Attrib
1 0 @F @F @F @F

@Var @RT(14)bMoveIdentDone @RT(0) @T @F @DT @RT(4)BOOL @RT(0) @T @T @BASIC 0 @F
@F @F
@T
@BEG_Attrib
3 @RT(5)FALSE @RT(0) @RT(0)
@END_Attrib
1 0 @F @F @F @F

@Var @RT(9)sFileName @RT(0) @T @F @DT @RT(11)STRING(255) @RT(0) @T @T @STRING 0 @F @RT(3)255 @F
@F @F
@T
@BEG_Attrib
3 @RT(0) @RT(0) @RT(0)
@END_Attrib
1 0 @F @F @F @F

@Var @RT(12)iFileCounter @RT(0) @T @F @DT @RT(5)UDINT @RT(0) @T @T @BASIC 0 @F
@F @F
@T
@BEG_Attrib
3 @RT(1)1 @RT(0) @RT(0)
@END_Attrib
1 0 @F @F @F @F

@Var @RT(11)ConstVisFwd @RT(0) @T @T @DERIVED 0 @T @T @DT @RT(8)tsVelPre @RT(0) @T @T @UNKNOWN 0 @F
@F @F
@T
@BEG_Attrib
3 @RT(0) @RT(41)const output for ejector forward movement @RT(0)
@END_Attrib
1 0 @F @F @F @F

@Var @RT(11)ConstVisBwd @RT(0) @T @T @DERIVED 0 @T @T @DT @RT(8)tsVelPre @RT(0) @T @T @UNKNOWN 0 @F
@F @F
@T
@BEG_Attrib
3 @RT(0) @RT(41)const output for ejector forward movement @RT(0)
@END_Attrib
1 0 @F @F @F @F

@Var @RT(12)bMinFwdRetry @RT(0) @T @F @DT @RT(4)BOOL @RT(0) @T @T @BASIC 0 @F
@F @F
@T
@BEG_Attrib
3 @RT(0) @RT(0) @RT(0)
@END_Attrib
1 0 @F @F @F @F

@Var @RT(12)bMinBwdRetry @RT(0) @T @F @DT @RT(4)BOOL @RT(0) @T @T @BASIC 0 @F
@F @F
@T
@BEG_Attrib
3 @RT(0) @RT(0) @RT(0)
@END_Attrib
1 0 @F @F @F @F

@Var @RT(15)bMinFwdDetected @RT(0) @T @F @DT @RT(4)BOOL @RT(0) @T @T @BASIC 0 @F
@F @F
@T
@BEG_Attrib
3 @RT(0) @RT(0) @RT(0)
@END_Attrib
1 0 @F @F @F @F

@Var @RT(15)bMinBwdDetected @RT(0) @T @F @DT @RT(4)BOOL @RT(0) @T @T @BASIC 0 @F
@F @F
@T
@BEG_Attrib
3 @RT(0) @RT(0) @RT(0)
@END_Attrib
1 0 @F @F @F @F

@Var @RT(9)sMoveName @RT(0) @T @F @DT @RT(10)STRING(32) @RT(0) @T @T @STRING 0 @F @RT(2)32 @F
@F @F
@T
@BEG_Attrib
3 @RT(0) @RT(0) @RT(0)
@END_Attrib
1 0 @F @F @F @F

@Var @RT(17)rMaxPressureLimit @RT(0) @T @F @DT @RT(4)REAL @RT(0) @T @T @BASIC 0 @F
@F @F
@T
@BEG_Attrib
3 @RT(5)150.0 @RT(0) @RT(0)
@END_Attrib
1 0 @F @F @F @F

@Var @RT(14)rRefSpeedLimit @RT(0) @T @F @DT @RT(4)REAL @RT(0) @T @T @BASIC 0 @F
@F @F
@T
@BEG_Attrib
3 @RT(0) @RT(0) @RT(0)
@END_Attrib
1 0 @F @F @F @F

@Var @RT(14)rSpeedLimitFwd @RT(0) @T @F @DT @RT(4)REAL @RT(0) @T @T @BASIC 0 @F
@F @F
@T
@BEG_Attrib
3 @RT(0) @RT(0) @RT(0)
@END_Attrib
1 0 @F @F @F @F

@Var @RT(14)rSpeedLimitBwd @RT(0) @T @F @DT @RT(4)REAL @RT(0) @T @T @BASIC 0 @F
@F @F
@T
@BEG_Attrib
3 @RT(0) @RT(0) @RT(0)
@END_Attrib
1 0 @F @F @F @F

@Var @RT(8)bTimeOut @RT(0) @T @F @DT @RT(4)BOOL @RT(0) @T @T @BASIC 0 @F
@F @F
@T
@BEG_Attrib
3 @RT(0) @RT(0) @RT(0)
@END_Attrib
1 0 @F @F @F @F

@Var @RT(13)bStopUnstable @RT(0) @T @F @DT @RT(4)BOOL @RT(0) @T @T @BASIC 0 @F
@F @F
@T
@BEG_Attrib
3 @RT(0) @RT(0) @RT(0)
@END_Attrib
1 0 @F @F @F @F

@Var @RT(12)dMaxMoveTime @RT(0) @T @F @DT @RT(4)TIME @RT(0) @T @T @BASIC 0 @F
@F @F
@T
@BEG_Attrib
3 @RT(0) @RT(0) @RT(0)
@END_Attrib
1 0 @F @F @F @F

@Var @RT(19)dMaxMoveTimeSaveFwd @RT(0) @T @F @DT @RT(4)TIME @RT(0) @T @T @BASIC 0 @F
@F @F
@T
@BEG_Attrib
3 @RT(0) @RT(0) @RT(0)
@END_Attrib
1 0 @F @F @F @F

@Var @RT(19)dMaxMoveTimeSaveBwd @RT(0) @T @F @DT @RT(4)TIME @RT(0) @T @T @BASIC 0 @F
@F @F
@T
@BEG_Attrib
3 @RT(0) @RT(0) @RT(0)
@END_Attrib
1 0 @F @F @F @F

@Var @RT(7)TimeOut @RT(0) @T @T @DERIVED 0 @T @T @DT @RT(3)TON @RT(0) @T @T @UNKNOWN 0 @F
@F @F
@T
@BEG_Attrib
3 @RT(0) @RT(0) @RT(0)
@END_Attrib
1 0 @F @F @F @F

@Var @RT(15)rMoveStrokeTime @RT(0) @T @F @DT @RT(4)REAL @RT(0) @T @T @BASIC 0 @F
@F @F
@T
@BEG_Attrib
3 @RT(0) @RT(0) @RT(0)
@END_Attrib
1 0 @F @F @F @F

@Var @RT(12)rStartFactor @RT(0) @T @F @DT @RT(4)REAL @RT(0) @T @T @BASIC 0 @F
@F @F
@T
@BEG_Attrib
3 @RT(3)0.1 @RT(0) @RT(0)
@END_Attrib
1 0 @F @F @F @F

@Var @RT(20)rMaxRefPressureLimit @RT(0) @T @F @DT @RT(4)REAL @RT(0) @T @T @BASIC 0 @F
@F @F
@T
@BEG_Attrib
3 @RT(0) @RT(0) @RT(0)
@END_Attrib
1 0 @F @F @F @F

@Var @RT(16)sWriteSpeedLimit @RT(0) @T @F @DT @RT(11)STRING(255) @RT(0) @T @T @STRING 0 @F @RT(3)255 @F
@F @F
@T
@BEG_Attrib
3 @RT(0) @RT(0) @RT(0)
@END_Attrib
1 0 @F @F @F @F

@Var @RT(14)dMoveTimeLimit @RT(0) @T @F @DT @RT(4)TIME @RT(0) @T @T @BASIC 0 @F
@F @F
@T
@BEG_Attrib
3 @RT(4)T#2m @RT(0) @RT(0)
@END_Attrib
1 0 @F @F @F @F

@Var @RT(16)bMoveTimeLimited @RT(0) @T @F @DT @RT(4)BOOL @RT(0) @T @T @BASIC 0 @F
@F @F
@T
@BEG_Attrib
3 @RT(0) @RT(0) @RT(0)
@END_Attrib
1 0 @F @F @F @F

@Var @RT(15)dMoveTimeOffset @RT(0) @T @F @DT @RT(4)TIME @RT(0) @T @T @BASIC 0 @F
@F @F
@T
@BEG_Attrib
3 @RT(4)T#5s @RT(0) @RT(0)
@END_Attrib
1 0 @F @F @F @F

@Var @RT(14)rStartPosition @RT(0) @T @F @DT @RT(4)REAL @RT(0) @T @T @BASIC 0 @F
@F @F
@T
@BEG_Attrib
3 @RT(0) @RT(0) @RT(0)
@END_Attrib
1 0 @F @F @F @F

@Var @RT(20)rMinMovementPosition @RT(0) @T @F @DT @RT(4)REAL @RT(0) @T @T @BASIC 0 @F
@F @F
@T
@BEG_Attrib
3 @RT(0) @RT(0) @RT(0)
@END_Attrib
1 0 @F @F @F @F

@Var @RT(18)rVelocitSizeFactor @RT(0) @T @F @DT @RT(4)REAL @RT(0) @T @T @BASIC 0 @F
@F @F
@T
@BEG_Attrib
3 @RT(3)1.0 @RT(0) @RT(0)
@END_Attrib
1 0 @F @F @F @F

@Var @RT(12)rMinStopRamp @RT(0) @T @F @DT @RT(4)REAL @RT(0) @T @T @BASIC 0 @F
@F @F
@T
@BEG_Attrib
3 @RT(3)1.0 @RT(0) @RT(0)
@END_Attrib
1 0 @F @F @F @F

@Var @RT(16)rMinStrokeFactor @RT(0) @T @F @DT @RT(4)REAL @RT(0) @T @T @BASIC 0 @F
@F @F
@T
@BEG_Attrib
3 @RT(3)2.0 @RT(0) @RT(0)
@END_Attrib
1 0 @F @F @F @F

@Var @RT(15)rMaxPressureFwd @RT(0) @T @F @DT @RT(4)REAL @RT(0) @T @T @BASIC 0 @F
@F @F
@T
@BEG_Attrib
3 @RT(0) @RT(0) @RT(0)
@END_Attrib
1 0 @F @F @F @F

@Var @RT(15)rMaxPressureBwd @RT(0) @T @F @DT @RT(4)REAL @RT(0) @T @T @BASIC 0 @F
@F @F
@T
@BEG_Attrib
3 @RT(0) @RT(0) @RT(0)
@END_Attrib
1 0 @F @F @F @F

@Var @RT(18)rPressureFactorFwd @RT(0) @T @F @DT @RT(4)REAL @RT(0) @T @T @BASIC 0 @F
@F @F
@T
@BEG_Attrib
3 @RT(0) @RT(0) @RT(0)
@END_Attrib
1 0 @F @F @F @F

@Var @RT(18)rPressureFactorBwd @RT(0) @T @F @DT @RT(4)REAL @RT(0) @T @T @BASIC 0 @F
@F @F
@T
@BEG_Attrib
3 @RT(0) @RT(0) @RT(0)
@END_Attrib
1 0 @F @F @F @F

@Var @RT(13)rPressureStep @RT(0) @T @F @DT @RT(4)REAL @RT(0) @T @T @BASIC 0 @F
@F @F
@T
@BEG_Attrib
3 @RT(3)5.0 @RT(0) @RT(0)
@END_Attrib
1 0 @F @F @F @F

@END_Dcl

@END_Export

@BEG_Export

@BEG_Algo
@POSTUPDATE_ALGORITHM @RT(17)pMinCommandListen @STRUCTURED_TEXT
@RT(0) @RT(72)sv_GlobalIdentMinSpeedStatus.Command,sv_GlobalIdentMinSpeedStatus.bStart @RT(9)PU_Task_7 @F @F
@END_Algo

@BEG_Dcl
@RT(16)DclTreeContainer
1
@Var @RT(1)i @RT(0) @T @F @DT @RT(4)DINT @RT(0) @T @T @BASIC 0 @F
@F @F
@T
@BEG_Attrib
3 @RT(0) @RT(0) @RT(0)
@END_Attrib
1 4 @F @F @F @F

@END_Dcl

@END_Export

@BEG_Export

@BEG_Algo
@PROCESS_ALGORITHM @RT(18)paMinCalibSequence @SEQUENTIAL_FLOW_CHART
@RT(0) @RT(0) @RT(7)TaskMid @F @F
@END_Algo

@BEG_Dcl
@RT(16)DclTreeContainer
6
@Var @RT(1)j @RT(0) @T @F @DT @RT(4)DINT @RT(0) @T @T @BASIC 0 @F
@F @F
@T
@BEG_Attrib
3 @RT(0) @RT(0) @RT(0)
@END_Attrib
1 4 @F @F @F @F

@Var @RT(1)i @RT(0) @T @F @DT @RT(4)DINT @RT(0) @T @T @BASIC 0 @F
@F @F
@T
@BEG_Attrib
3 @RT(0) @RT(0) @RT(0)
@END_Attrib
1 4 @F @F @F @F

@Var @RT(12)tmpMovements @RT(0) @T @T @DERIVED 0 @T @T @DT @RT(21)tyIdentSpeedMovements @RT(0) @T @T @UNKNOWN 0 @F
@F @F
@T
@BEG_Attrib
3 @RT(0) @RT(0) @RT(0)
@END_Attrib
1 0 @F @F @F @F

@Var @RT(13)iMaxMovements @RT(0) @T @F @DT @RT(4)DINT @RT(0) @T @T @BASIC 0 @F
@F @F
@T
@BEG_Attrib
3 @RT(0) @RT(0) @RT(0)
@END_Attrib
1 0 @F @F @F @F

@Var @RT(4)tmpM @RT(0) @T @T @DERIVED 0 @T @T @DT @RT(20)tpIdentSpeedMovement @RT(0) @T @T @UNKNOWN 0 @F
@F @F
@T
@BEG_Attrib
3 @RT(0) @RT(0) @RT(0)
@END_Attrib
1 0 @F @F @F @F

@Var @RT(11)ConstBwdVis @RT(0) @T @T @DERIVED 0 @T @T @DT @RT(8)tsVelPre @RT(0) @T @T @UNKNOWN 0 @F
@F @F
@T
@BEG_Attrib
3 @RT(0) @RT(0) @RT(0)
@END_Attrib
1 0 @F @F @F @F

@END_Dcl

@END_Export

@BEG_Export

@BEG_Algo
@POSTUPDATE_ALGORITHM @RT(10)pDataState @STRUCTURED_TEXT
@RT(0) @RT(12)sv_DataState @RT(10)PU_Task_13 @F @F
@END_Algo

@BEG_Dcl
@RT(16)DclTreeContainer
2
@Var @RT(20)bMDLoadingInProgress @RT(0) @T @F @DT @RT(4)BOOL @RT(0) @T @T @BASIC 0 @F
@F @F
@T
@BEG_Attrib
3 @RT(0) @RT(35)loading of machine data in progress @RT(0)
@END_Attrib
1 0 @F @F @F @F

@Var @RT(1)i @RT(0) @T @F @DT @RT(4)DINT @RT(0) @T @T @BASIC 0 @F
@F @F
@T
@BEG_Attrib
3 @RT(0) @RT(0) @RT(0)
@END_Attrib
1 4 @F @F @F @F

@END_Dcl

@END_Export

@BEG_Body
@TL(62)
(**************************************** WARNING ********************************************
 *** The KEBA Kemro K2 System including software is not intended for safety control tasks! ***
 ***                       For further information see Comment tab!                        ***
 *********************************************************************************************)

i := 1;

rpPosition := GET_SYNC_REFTO('Ejector1.ai_Position', T#0s, Status);
IF Status = KSYS_Status_OK THEN
    sv_GlobalIdentMaxSpeedStatus.pMovements[i] := @sv_EjectorIdentMaxMovement;
    sv_GlobalIdentMinSpeedStatus.pMovements[i] := @sv_EjectorIdentMinMovement;
    i := i + 1;
END_IF;

sv_GlobalIdentMaxSpeedStatus.pMovements[i] := @sv_MoldIdentMaxMovement;
sv_GlobalIdentMinSpeedStatus.pMovements[i] := @sv_MoldIdentMinMovement;
i := i + 1;

pOption := GET_SYNC_REFTO('Nozzle1.sv_Options', T#0s, Status);
IF (Status = KSYS_Status_OK) AND ((pOption^ AND cOptionHydraulic) = cOptionHydraulic) THEN;
    //hydraulic nozzle -> check if ai_Position is available
    rpPosition := GET_SYNC_REFTO('Nozzle1.ai_Position', T#0s, Status);
    IF Status = KSYS_Status_OK THEN
        sv_GlobalIdentMaxSpeedStatus.pMovements[i] := @sv_NozzleIdentMaxMovement;
        sv_GlobalIdentMinSpeedStatus.pMovements[i] := @sv_NozzleIdentMinMovement;
        i := i + 1;
    END_IF;
END_IF;

sv_GlobalIdentMaxSpeedStatus.pMovements[i] := @sv_InjectionIdentMaxMovement;
sv_GlobalIdentMinSpeedStatus.pMovements[i] := @sv_InjectionIdentMinMovement;
i := i + 1;

(* sort them by iOrder *)
FOR k := 1 TO i - 2 DO
    FOR j := 1 TO i - 1 - k DO
        IF sv_GlobalIdentMaxSpeedStatus.pMovements[j]^.iOrder > sv_GlobalIdentMaxSpeedStatus.pMovements[j + 1]^.iOrder THEN
            tmpM := sv_GlobalIdentMaxSpeedStatus.pMovements[j];
            sv_GlobalIdentMaxSpeedStatus.pMovements[j] := sv_GlobalIdentMaxSpeedStatus.pMovements[j + 1];
            sv_GlobalIdentMaxSpeedStatus.pMovements[j + 1] := tmpM;
            tmpM := sv_GlobalIdentMinSpeedStatus.pMovements[j];
            sv_GlobalIdentMinSpeedStatus.pMovements[j] := sv_GlobalIdentMinSpeedStatus.pMovements[j + 1];
            sv_GlobalIdentMinSpeedStatus.pMovements[j + 1] := tmpM;
        END_IF;
    END_FOR;
END_FOR;

sv_GlobalIdentMaxSpeedStatus.iMaxStep := i - 1;
sv_GlobalIdentMinSpeedStatus.iMaxStep := i - 1;

sv_GlobalIdentMaxSpeedStatus.iCurrentStep := 0;
sv_GlobalIdentMaxSpeedStatus.Status := tnCalibState_None;
sv_GlobalIdentMaxSpeedStatus.bInitDone := TRUE;

sv_GlobalIdentMinSpeedStatus.iCurrentStep := 0;
sv_GlobalIdentMinSpeedStatus.Status := tnCalibState_None;
sv_GlobalIdentMinSpeedStatus.bInitDone := TRUE;

STOP_PROCESS_ALGORITHM();

@END_Body

@@@BEG_Comment@@@
@TL(0)

@@@END_Comment@@@

@BEG_Body
@TL(20)
IF ((sv_GlobalIdentMaxSpeedStatus.Status = tnCalibState_Running) OR (sv_GlobalIdentMinSpeedStatus.Status = tnCalibState_Running)) AND
    (sv_iPendingAlarms <> 0) THEN

   dummy := Print('auto max. speed identification stopped because alarms of class 1/2/3 pending');

   //trace all pending alarms
   fbTracePendingAlarms();

   IF (sv_GlobalIdentMaxSpeedStatus.Status = tnCalibState_Running) THEN
      sv_GlobalIdentMaxSpeedStatus.Command := tnCalibCommand_Stop;
      sv_GlobalIdentMaxSpeedStatus.Status := tnCalibState_Aborted;
   ELSE
      sv_GlobalIdentMinSpeedStatus.Command := tnCalibCommand_Stop;
      sv_GlobalIdentMinSpeedStatus.Status := tnCalibState_Aborted;
   END_IF;

   SET_ALARM(Name := erCalibrationSpeedStopped,
             Param1 := miErrorNo);
END_IF;

@END_Body

@@@BEG_Comment@@@
@TL(0)

@@@END_Comment@@@

@BEG_Body
@TL(15)
IF mbprActPressureLinked THEN
   rActPressure := mprActPressure^;
ELSE
   rActPressure := 0.0;
END_IF;
abSpeedMeasure.aMeasure(bRestart := mbRestartMeas,
                        rPosition := mActMovement^.prPosition^,
                        rRefVelocity := mrRefVelocity,
                        rActVelocity := mActMovement^.prActVelocity^,
                        rRefPressure := mrRefPressure,
                        rActPressure := rActPressure,
                        rMaxLimitPosition := mrMaxLimitPosition,
                        rMinLimitPosition := mrMinLimitPosition);
mbRestartMeas := FALSE;

@END_Body

@@@BEG_Comment@@@
@TL(0)

@@@END_Comment@@@

@BEG_Body
@TL(2)
aMeasure();

@END_Body

@@@BEG_Comment@@@
@TL(0)

@@@END_Comment@@@

@BEG_Body
@TL(2)
aMeasure();

@END_Body

@@@BEG_Comment@@@
@TL(0)

@@@END_Comment@@@

@BEG_Body
@TL(5)
mbRestartMeas := TRUE;
abSpeedMeasure.aReset();
abSpeedMeasure.aMeasure(bRestart := TRUE);
START_PROCESS_ALGORITHM(paMeasureMid);

@END_Body

@@@BEG_Comment@@@
@TL(0)

@@@END_Comment@@@

@BEG_Body
@TL(4)
STOP_PROCESS_ALGORITHM(paMeasureMid);
abSpeedMeasure.aCloseMeasure();

@END_Body

@@@BEG_Comment@@@
@TL(0)

@@@END_Comment@@@

@BEG_Body
@TL(7)
mbLogFileSaved := FALSE;
msFileName := sFileName;
miFileCounter := iFileCounter;
mbDeleteFiles := bDeleteFiles;

START_PROCESS_ALGORITHM(paWriteLog);

@END_Body

@@@BEG_Comment@@@
@TL(0)

@@@END_Comment@@@

@BEG_Body
@TL(14)
fbIdentWriteLog(sFileName    := msFileName,
                iFileCounter := miFileCounter,
                bDeleteFiles := mbDeleteFiles,
                rMaxVelocity := mrMaxVelocity,
                rMaxPressure := mrMaxPressure,
                bVelocityLimitReached := mbVelocityLimitReached,
                bPressureLimitReached := mbPressureLimitReached);
IF fbIdentWriteLog.bDone THEN
   mbLogFileSaved := TRUE;
ELSE
   mbLogFileSaved := FALSE;
END_IF;
STOP_PROCESS_ALGORITHM();

@END_Body

@@@BEG_Comment@@@
@TL(0)

@@@END_Comment@@@

@BEG_Body
@TL(18)
IF mActMovement^.bPositionIncreasingFwd THEN
   mActMovement^.prIdentPosition^ := mActMovement^.prStroke^ * mrMaxPositionFactor;
ELSE
   mActMovement^.prIdentPosition^ := mActMovement^.prStroke^ * mrMinPositionFactor;
END_IF;
mActMovement^.pbMoveIdent^ := TRUE;

evStartRequestData.DeviceId := mActMovement^.DeviceId;
evStartRequestData.MoveDir := cMoveFwd;
IF mActMovement^.MoveId > cMoveNone THEN
   evStartRequestData.MoveId := mActMovement^.MoveId;
ELSE
   evStartRequestData.MoveId := cMoveFwd;
END_IF;

SET_EVENT(evStartRequest, evStartRequestData);

@END_Body

@@@BEG_Comment@@@
@TL(0)

@@@END_Comment@@@

@BEG_Body
@TL(18)
IF mActMovement^.bPositionIncreasingFwd THEN
   mActMovement^.prIdentPosition^ := mActMovement^.prStroke^ * mrMinPositionFactor;
ELSE
   mActMovement^.prIdentPosition^ := mActMovement^.prStroke^ * mrMaxPositionFactor;
END_IF;
mActMovement^.pbMoveIdent^ := TRUE;

evStartRequestData.DeviceId := mActMovement^.DeviceId;
evStartRequestData.MoveDir := cMoveBwd;
IF mActMovement^.MoveId > cMoveNone THEN
   evStartRequestData.MoveId := cMoveDecompAftPlast;
ELSE
   evStartRequestData.MoveId := cMoveBwd;
END_IF;

SET_EVENT(evStartRequest, evStartRequestData);

@END_Body

@@@BEG_Comment@@@
@TL(0)

@@@END_Comment@@@

@BEG_Body
@TL(11)
evStopRequestData.DeviceId := mActMovement^.DeviceId;
evStopRequestData.MoveDir := cMoveFwd;
evStopRequestData.MoveId := cMoveFwd;
SET_EVENT(evStopRequest, evStopRequestData);
mActMovement^.pbMoveIdent^ := FALSE;
mActMovement^.prIdentPosition^ := 0.0;
mActMovement^.prStopRamp^ := 0.0;

@END_Body

@@@BEG_Comment@@@
@TL(0)

@@@END_Comment@@@

@BEG_Body
@TL(14)
evStopRequestData.DeviceId := mActMovement^.DeviceId;
evStopRequestData.MoveDir := cMoveBwd;
IF mActMovement^.MoveId > cMoveNone THEN
   evStopRequestData.MoveId := cMoveDecompAftPlast;
ELSE
   evStopRequestData.MoveId := cMoveBwd;
END_IF;
SET_EVENT(evStopRequest, evStopRequestData);
mActMovement^.pbMoveIdent^ := FALSE;
mActMovement^.prIdentPosition^ := 0.0;
mActMovement^.prStopRamp^ := 0.0;

@END_Body

@@@BEG_Comment@@@
@TL(0)

@@@END_Comment@@@

@BEG_Body
@TL(7)
sv_GlobalIdentMinSpeedStatus.Status := tnCalibState_Aborted;
mActMovement^.Status := tnCalibState_Error;

dummy := Print('Calib movement "%s" aborted.', sMovementName);

@END_Body

@@@BEG_Comment@@@
@TL(0)

@@@END_Comment@@@

@BEG_Body
@TL(63)
IF (bUsePressureMode) THEN
   IF (rMaxActSpeed = 0.0) THEN
      rMaxActSpeed := rMaxSpeedLimit;
   END_IF;
   IF (bPresLimitReached) THEN
      // reduce refernce value
      rMaxActSpeed := rActSpeedLimit;
      IF (ABS(rMaxActSpeed - rMinActSpeed) < rMinSpeedDifference * rMaxSpeedLimit) THEN
         bMaxDetected := TRUE;
         rMaxSpeed := rMinActSpeed;
         rMinActSpeed := 0.0;
         rMaxActSpeed := 0.0;
      ELSE
         bMaxDetected := FALSE;
         rRefSpeed := 0.5 * (rMaxActSpeed + rMinActSpeed);
      END_IF;
   ELSE
      // ccompare with old value
      IF (rActSpeedLimit = rMaxSpeedLimit) THEN // maximum used at start
         // maximum with tolerance reached
         bMaxDetected := TRUE;
         rMaxSpeed := rMaxSpeedLimit;
         rMinActSpeed := 0.0;
         rMaxActSpeed := 0.0;
      ELSE
         // increase
         rMinActSpeed := rActSpeedLimit;
         IF (ABS(rMaxActSpeed - rMinActSpeed) < rMinSpeedDifference * rMaxSpeedLimit) THEN
            bMaxDetected := TRUE;
            rMaxSpeed := rMinActSpeed;
            rMinActSpeed := 0.0;
            rMaxActSpeed := 0.0;
         ELSE
            rRefSpeed := 0.5 * (rMaxActSpeed + rMinActSpeed);
         END_IF;
      END_IF;
   END_IF;
ELSE
   IF (rActSpeedLimit = rMaxSpeedLimit) THEN // maximum used at start
      IF (rActMaxSpeed > rSpeedReachedFactor * rActSpeedLimit)  THEN
      // maximum with tolerance reached
         bMaxDetected := TRUE;
         rMaxSpeed := rMaxSpeedLimit;
      ELSE
      // actual speed lower than maximum with tolerance
         bMaxDetected := FALSE;
         rRefSpeed := rActMaxSpeed;
         rMaxActSpeed := rActMaxSpeed;
      END_IF;
   ELSE
      IF (rActMaxSpeed > rSpeedReachedFactor * rActSpeedLimit) THEN
      // reference speed with tolerance reached
         bMaxDetected := TRUE;
         rMaxSpeed := rRefSpeed;
      ELSE
      // actual speed lower than reference speed with tolerance reached
      // check calibration of pump/valve
         bMaxDetected := TRUE;
         rMaxSpeed := rRefSpeed;
      END_IF;
   END_IF;
END_IF;

@END_Body

@@@BEG_Comment@@@
@TL(0)

@@@END_Comment@@@

@BEG_Body
@TL(4)

START_PROCESS_ALGORITHM(paRedoMax);

@END_Body

@@@BEG_Comment@@@
@TL(0)

@@@END_Comment@@@

@BEG_Body
@TL(26)
bIdentActive := FALSE;
FOR i:= 1 TO cCalibMovements DO
   IF CHECK_REF(sv_GlobalIdentMaxSpeedStatus.pMovements[i]^) THEN
      IF sv_GlobalIdentMaxSpeedStatus.pMovements[i]^.bRedo THEN
         mActMovement := sv_GlobalIdentMaxSpeedStatus.pMovements[i];
         bIdentActive := TRUE;
         sv_GlobalIdentMaxSpeedStatus.iCurrentStep :=  i;
         mCalibCounter := i;
         IF sv_OperationMode = nSetup THEN
            mbUseSingleMovement := TRUE;
            START_PROCESS_ALGORITHM(paMaxSingleMovement);
         ELSE
            sv_GlobalIdentMaxSpeedStatus.pMovements[i]^.bRedo := FALSE;
            SET_ALARM(erSetupModeRequiredForCalib);
         END_IF;
         EXIT;
      END_IF;
   END_IF;
END_FOR;
IF ((NOT bIdentActive) AND (sv_GlobalIdentMaxSpeedStatus.Status = tnCalibState_Running)) THEN
   sv_GlobalIdentMaxSpeedStatus.Status := tnCalibState_Aborted;
END_IF;

STOP_PROCESS_ALGORITHM();

@END_Body

@@@BEG_Comment@@@
@TL(0)

@@@END_Comment@@@

@BEG_SfcBody
42 49 48

@BEG_SfcData 2
@StepSeq @RT(4)sseq @F 39
@Step @RT(7)S_RESET @F @F @T @F @RT(0) @F
@AcbCont @RT(7)unnamed @F 0

@Trans @RT(7)Trans47 @F @T @F @F @T @T @TL(2)
mbLogFileSaved

@RT(7)Trans47 @F
@Step @RT(6)S_STOP @F @F @F @F @RT(0) @F
@AcbCont @RT(7)unnamed @F 1
@Acb @RT(9)AStopSelf @F @T @RT(1)P @RT(0) @F @F @T @TL(12)
sv_GlobalIdentMaxSpeedStatus.Command := tnCalibCommand_None;
sv_bAutoIdentRunning := FALSE;
mActMovement^.bRedo := FALSE;
mActMovement^.prStopRamp^ := 0.0;
mActMovement^.pConstFwdVis^ := ConstVisFwd;
mActMovement^.pConstBwdVis^ := ConstVisBwd;

//release memory
abSpeedMeasure.aEnd();

STOP_PROCESS_ALGORITHM();

@F

@Trans @RT(8)TRestart @F @T @F @F @T @T @TL(2)
TRUE

@RT(8)TRestart @F
@Step @RT(6)S_INIT @F @T @F @F @RT(0) @F
@AcbCont @RT(7)unnamed @F 1
@Acb @RT(7)Action3 @F @T @RT(1)P @RT(0) @F @F @T @TL(43)
miErrorNo := 0;

ConstVisFwd := mActMovement^.pConstFwdVis^;
ConstVisBwd := mActMovement^.pConstBwdVis^;

sv_GlobalIdentMaxSpeedStatus.Status := tnCalibState_Running;
mActMovement^.Status := tnCalibState_Running;
sMoveName := mActMovement^.sName;

abSpeedMeasure.aInit();

bMaxFwdRetry := FALSE;
bMaxBwdRetry := FALSE;

IF (mActMovement^.rMaxPositionLimitFactor > mActMovement^.rMinPositionLimitFactor) AND
   (mActMovement^.rMinPositionLimitFactor > 0.0) AND (mActMovement^.rMaxPositionLimitFactor < 1.0) THEN
   mrMaxPositionFactor := mActMovement^.rMaxPositionLimitFactor;
   mrMinPositionFactor := mActMovement^.rMinPositionLimitFactor;
ELSE // use deafult values
   mrMaxPositionFactor := 0.8;
   mrMinPositionFactor := 0.2;
END_IF;

mprActPressure := sv_PumpData[mActMovement^.DeviceId.IndexId].prActSysPressure;
IF CHECK_REF(mprActPressure^) THEN
   mbprActPressureLinked := TRUE;
ELSE
   mbprActPressureLinked := FALSE;
END_IF;

IF CHECK_REF(mActMovement^.pdDelayTimeOffFwd^) THEN
   bDelayTimeOffFwdLinked := TRUE;
   dDelayTimeOffFwd := mActMovement^.pdDelayTimeOffFwd^;
ELSE
   bDelayTimeOffFwdLinked := FALSE;
END_IF;
IF CHECK_REF(mActMovement^.pdDelayTimeOffBwd^) THEN
   bDelayTimeOffBwdLinked := TRUE;
   dDelayTimeOffBwd := mActMovement^.pdDelayTimeOffBwd^;
ELSE
   bDelayTimeOffBwdLinked := FALSE;
END_IF;

@F

@Trans @RT(13)TMoveStartBwd @F @T @F @F @T @T @TL(3)
TRUE

@RT(13)TMoveStartBwd @F
@Step @RT(14)S_MoveStartBwd @F @F @F @F @RT(0) @F
@AcbCont @RT(7)unnamed @F 3
@Acb @RT(13)AMoveStartBwd @F @T @RT(1)P @RT(0) @F @F @T @TL(4)
bMoveBwdDone := FALSE;
miErrorNo := cIdentSpeedMaxBwdInit;
aStartMovementBwd();

@F
@Acb @RT(23)ACheckMoveStartBwdReady @F @T @RT(1)N @RT(0) @F @F @T @TL(5)
fbCheckReady(DeviceId := evStartRequestData.DeviceId);
IF fbCheckReady.bReady THEN
   bMoveBwdDone := TRUE;
END_IF;

@F
@Acb @RT(18)AMoveStartBwdReady @F @T @RT(2)P0 @RT(0) @F @F @T @TL(2)
aStopMovementBwd();

@F

@AltBranch @RT(3)alt @F 2
@TransSeq @RT(4)tseq @F 1
@Trans @RT(8)TInitBwd @F @T @F @F @T @T @TL(2)
bMoveBwdDone

@RT(8)TInitBwd @F

@TransSeq @RT(4)tseq @F 4
@Trans @RT(17)TStopMoveStartBwd @F @T @F @F @T @F @TL(5)
sv_GlobalIdentMaxSpeedStatus.Status = tnCalibState_Aborted OR
sv_GlobalIdentMaxSpeedStatus.Status = tnCalibState_None
OR sv_iPendingAlarms <> 0
OR mActMovement^.bRedo = FALSE

@RT(17)TStopMoveStartBwd @F
@Step @RT(18)S_StopMoveStartBwd @F @F @T @F @RT(0) @F
@AcbCont @RT(7)unnamed @F 1
@Acb @RT(17)AStopMoveStartBwd @F @T @RT(1)P @RT(0) @F @F @T @TL(2)
aStopMovementError(sMovementName := CONCAT(sMoveName, ' max ident Fwd: Bwd to initial position'));

@F

@Trans @RT(6)TReset @F @T @F @F @T @F @TL(2)
TRUE

@RT(6)TReset @F
@Goto @RT(7)S_RESET @F @F

@Step @RT(22)S_CHECK_ALARMS_INITBWD @F @F @F @F @RT(0) @F
@AcbCont @RT(7)unnamed @F 0

@AltBranch @RT(3)alt @F 2
@TransSeq @RT(4)tseq @F 1
@Trans @RT(11)TStartIdent @F @T @F @F @T @T @TL(2)
S_CHECK_ALARMS_INITBWD.T > T#100ms

@RT(11)TStartIdent @F

@TransSeq @RT(4)tseq @F 2
@Trans @RT(12)TStopInitBwd @F @T @F @F @T @F @TL(2)
sv_iPendingAlarms <> 0

@RT(12)TStopInitBwd @F
@Goto @RT(18)S_StopMoveStartBwd @F @F

@Step @RT(15)S_INITCALIB_FWD @F @F @F @F @RT(0) @F
@AcbCont @RT(7)unnamed @F 1
@Acb @RT(13)aInitIdentFwd @F @T @RT(1)P @RT(0) @F @F @T @TL(18)
iFileCounter := 1;
IF (CHECK_REF(mActMovement^.prSizeFactorFwd^)) THEN
   IF (mActMovement^.prSizeFactorFwd^ > 0.0) THEN
      rVelocitSizeFactor := mActMovement^.prSizeFactorFwd^;
   END_IF;
ELSE
   rVelocitSizeFactor := 1.0;
END_IF;
rRefSpeedLimit := mActMovement^.prVelocityLimitFwd^;
rMaxPressureLimit := mActMovement^.prMaxPressureFwd^;
IF CHECK_REF(mActMovement^.prMaxPressureFwdHydr^) THEN
   rMaxRefPressureLimit := mActMovement^.prMaxPressureFwdHydr^;
ELSE
   rMaxRefPressureLimit := rMaxPressureLimit;
END_IF;

dummy := Print('Calib max speed %s Fwd started', sMoveName);

@F

@Trans @RT(7)TDelay1 @F @T @F @F @T @T @TL(2)
S_INITCALIB_FWD.T>T#1s

@RT(7)TDelay1 @F
@Step @RT(11)S_CALIB_FWD @F @F @T @F @RT(0) @F
@AcbCont @RT(7)unnamed @F 4
@Acb @RT(8)ADoCalib @F @T @RT(1)P @RT(0) @F @F @T @TL(52)
(* start calibration *)
// save actual settings
ConstVis := mActMovement^.pConstFwdVis^;

mActMovement^.pConstFwdVis^.Velocity.Output.rOutputValue := rRefSpeedLimit * rVelocitSizeFactor;
mActMovement^.pConstFwdVis^.Velocity.rMinOutput := 0.0;
mActMovement^.pConstFwdVis^.Pressure.Output.rOutputValue := MAX(mActMovement^.pConstFwdVis^.Pressure.Output.rOutputValue, rMaxPressureLimit);
mActMovement^.pConstFwdVis^.Pressure.Output.rRamp := MAX(1.0e9,ConstVis.Pressure.Output.rRamp);
IF mActMovement^.bPositionIncreasingFwd THEN
   mActMovement^.prIdentPosition^ := mActMovement^.prStroke^ * mrMaxPositionFactor;
   mrMinLimitPosition := rStartFactor * mActMovement^.prIdentPosition^ + (1.0 - rStartFactor) * mActMovement^.prPosition^;
   IF (mActMovement^.prIdentPosition^ - mActMovement^.prPosition^) > 0.0 THEN
      rMinStopRamp := rMinStrokeFactor * rRefSpeedLimit  * rRefSpeedLimit/ ABS(mActMovement^.prIdentPosition^ - mActMovement^.prPosition^);
   ELSE
      rMinStopRamp := 0.0;
   END_IF;
   mActMovement^.prStopRamp^ := MAX(mActMovement^.pConstFwdVis^.Velocity.Output.rRamp, rMinStopRamp);
   mrMaxLimitPosition := mActMovement^.prIdentPosition^;
ELSE
   mActMovement^.prIdentPosition^ := mActMovement^.prStroke^ * mrMinPositionFactor;
   mrMaxLimitPosition := (1.0 - rStartFactor) * mActMovement^.prPosition^ + rStartFactor * mActMovement^.prIdentPosition^;
   IF (mActMovement^.prPosition^ - mActMovement^.prIdentPosition^) > 0.0 THEN
      rMinStopRamp := rMinStrokeFactor * rRefSpeedLimit * rRefSpeedLimit / ABS(mActMovement^.prIdentPosition^ - mActMovement^.prPosition^);
   ELSE
      rMinStopRamp := 0.0;
   END_IF;
   mActMovement^.prStopRamp^ := MAX(mActMovement^.pConstFwdVis^.Velocity.Output.rRamp, rMinStopRamp);
   mrMinLimitPosition := mActMovement^.prIdentPosition^;
END_IF;
mActMovement^.pbMoveIdent^ := TRUE;
bMoveIdentDone := FALSE;

bMaxFwdDetected := FALSE;

mrRefVelocity := rRefSpeedLimit;
mrRefPressure := rMaxRefPressureLimit;
mbRestartMeas := TRUE;

IF bDelayTimeOffFwdLinked THEN
   mActMovement^.pdDelayTimeOffFwd^ := MAX(mActMovement^.pdDelayTimeOffFwd^, dMinDelayTimeOff);
END_IF;
IF bDelayTimeOffBwdLinked THEN
   mActMovement^.pdDelayTimeOffBwd^ := MAX(mActMovement^.pdDelayTimeOffBwd^, dMinDelayTimeOff);
END_IF;

aStartMeasurement();

sWriteSpeedLimit := REAL_TO_STRING(rRefSpeedLimit);
dummy := Print('Calib max output: act. max speed: %s', sWriteSpeedLimit);
miErrorNo := cIdentSpeedMaxFwdIdent;

@F
@Acb @RT(17)AStartMovementFwd @F @T @RT(1)P @RT(0) @F @F @T @TL(9)
evStartRequestData.DeviceId := mActMovement^.DeviceId;
evStartRequestData.MoveDir := cMoveFwd;
IF mActMovement^.MoveId > cMoveNone THEN
   evStartRequestData.MoveId := mActMovement^.MoveId;
ELSE
   evStartRequestData.MoveId := cMoveFwd;
END_IF;
SET_EVENT(evStartRequest, evStartRequestData);

@F
@Acb @RT(25)ACheckActMovementFwdReady @F @T @RT(1)N @RT(0) @F @F @T @TL(5)
fbCheckReady(DeviceId := evStartRequestData.DeviceId);
IF fbCheckReady.bReady THEN
   bMoveIdentDone := TRUE;
END_IF;

@F
@Acb @RT(16)AStopMovementFwd @F @T @RT(2)P0 @RT(0) @F @F @T @TL(15)
aStopMeasurement();
aStopMovementFwd();

mActMovement^.pConstFwdVis^ := ConstVis;
mActMovement^.prStopRamp^ := 0.0;

IF bDelayTimeOffFwdLinked THEN
   mActMovement^.pdDelayTimeOffFwd^ := dDelayTimeOffFwd;
END_IF;
IF bDelayTimeOffBwdLinked THEN
   mActMovement^.pdDelayTimeOffBwd^ := dDelayTimeOffBwd;
END_IF;

@F

@AltBranch @RT(3)alt @F 2
@TransSeq @RT(4)tseq @F 1
@Trans @RT(17)TMoveIdentFwdDone @F @T @F @F @T @T @TL(2)
bMoveIdentDone

@RT(17)TMoveIdentFwdDone @F

@TransSeq @RT(4)tseq @F 4
@Trans @RT(13)TStopIdentFwd @F @T @F @F @T @F @TL(5)
sv_GlobalIdentMaxSpeedStatus.Status = tnCalibState_Aborted OR
sv_GlobalIdentMaxSpeedStatus.Status = tnCalibState_None
OR sv_iPendingAlarms <> 0
OR mActMovement^.bRedo = FALSE

@RT(13)TStopIdentFwd @F
@Step @RT(14)S_StopIdentFwd @F @F @T @F @RT(0) @F
@AcbCont @RT(7)unnamed @F 1
@Acb @RT(13)AStopIdentFwd @F @T @RT(1)P @RT(0) @F @F @T @TL(2)
aStopMovementError(sMovementName := CONCAT(sMoveName, ' max ident Fwd'));

@F

@Trans @RT(7)TReset1 @F @T @F @F @T @F @TL(2)
TRUE

@RT(7)TReset1 @F
@Goto @RT(7)S_RESET @F @F

@Step @RT(18)S_CHECK_ALARMS_FWD @F @F @F @F @RT(0) @F
@AcbCont @RT(7)unnamed @F 0

@AltBranch @RT(3)alt @F 2
@TransSeq @RT(4)tseq @F 1
@Trans @RT(14)TStartWriteFwd @F @T @F @F @T @T @TL(2)
S_CHECK_ALARMS_FWD.T > T#100ms

@RT(14)TStartWriteFwd @F

@TransSeq @RT(4)tseq @F 2
@Trans @RT(14)TStopIdentFwd2 @F @T @F @F @T @F @TL(2)
sv_iPendingAlarms <> 0

@RT(14)TStopIdentFwd2 @F
@Goto @RT(14)S_StopIdentFwd @F @F

@Step @RT(11)S_WRITE_FWD @F @F @F @F @RT(0) @F
@AcbCont @RT(7)unnamed @F 1
@Acb @RT(9)AWriteFwd @F @T @RT(1)P @RT(0) @F @F @T @TL(11)
abSpeedMeasure.aGetMaxValues(rMaxSpeed => mrMaxVelocity,
                             rMaxPressure => mrMaxPressure,
                             bPressureLimitReached => mbPressureLimitReached,
                             bSpeedLimitReached => mbVelocityLimitReached);
sFileName := CONCAT(sMoveName,"_MAXSPEED_FWD_");
aWriteLog(sFileName := sFileName,
          iFileCounter := iFileCounter,
          bDeleteFiles := TRUE);
iFileCounter := iFileCounter + 1;

@F

@AltBranch @RT(3)alt @F 2
@TransSeq @RT(4)tseq @F 1
@Trans @RT(9)TWriteFwd @F @T @F @F @T @T @TL(2)
mbLogFileSaved

@RT(9)TWriteFwd @F

@TransSeq @RT(4)tseq @F 4
@Trans @RT(16)TAbortedWriteFwd @F @T @F @F @T @F @TL(2)
sv_GlobalIdentMaxSpeedStatus.Status = tnCalibState_Aborted

@RT(16)TAbortedWriteFwd @F
@Step @RT(17)S_AbortedWriteFwd @F @F @F @F @RT(0) @F
@AcbCont @RT(7)unnamed @F 1
@Acb @RT(16)AAbortedWriteFwd @F @T @RT(1)P @RT(0) @F @F @T @TL(3)
mActMovement^.Status := tnCalibState_Error;

@F

@Trans @RT(21)TResetAbortedWriteFwd @F @T @F @F @T @F @TL(2)
TRUE

@RT(21)TResetAbortedWriteFwd @F
@Goto @RT(7)S_RESET @F @F

@Step @RT(20)S_CHECK_MAXSPEED_FWD @F @F @F @F @RT(0) @F
@AcbCont @RT(7)unnamed @F 1
@Acb @RT(17)ACheckMaxSpeedFwd @F @T @RT(1)P @RT(0) @F @F @T @TL(18)
aCalcMaxSpeedOutput(rMaxSpeedLimit := mActMovement^.prVelocityLimitFwd^,
                    rActSpeedLimit := rRefSpeedLimit,
                    rActMaxSpeed := abSpeedMeasure.aGetMaxValues.rMaxSpeed,
                    bPresLimitReached := abSpeedMeasure.aGetMaxValues.bPressureLimitReached,
                    bUsePressureMode := (mrMaxPressure > 0.0));
bMaxFwdDetected := aCalcMaxSpeedOutput.bMaxDetected;
IF (bMaxFwdDetected) THEN
   rSpeedLimitFwd := rRefSpeedLimit;
   dummy := Print('Calib max output %s Fwd finished: max speed fwd = %f$N', sMoveName, rSpeedLimitFwd);
ELSE
   IF abSpeedMeasure.aGetMaxValues.bPressureLimitReached THEN
      sWriteSpeedLimit := REAL_TO_STRING(rRefSpeedLimit);
      dummy := Print('Calib max output: pressure limit reached with act. max speed %s', sWriteSpeedLimit);
   END_IF;
   bMaxFwdRetry := TRUE;
   rRefSpeedLimit := aCalcMaxSpeedOutput.rRefSpeed;
END_IF;

@F

@AltBranch @RT(3)alt @F 2
@TransSeq @RT(4)tseq @F 1
@Trans @RT(15)TMaxFwdDetected @F @T @F @F @T @T @TL(2)
bMaxFwdDetected

@RT(15)TMaxFwdDetected @F

@TransSeq @RT(4)tseq @F 6
@Trans @RT(7)Trans15 @F @T @F @F @T @T @TL(2)
bMaxFwdRetry

@RT(7)Trans15 @F
@Step @RT(13)S_MaxFwdRetry @F @F @F @F @RT(0) @F
@AcbCont @RT(7)unnamed @F 3
@Acb @RT(20)AStartMovementFwdBwd @F @T @RT(1)P @RT(0) @F @F @T @TL(4)
bMoveBwdDone := FALSE;
miErrorNo := cIdentSpeedMaxFwdStart;
aStartMovementBwd();

@F
@Acb @RT(28)ACheckActMovementFwdBwdReady @F @T @RT(1)N @RT(0) @F @F @T @TL(5)
fbCheckReady(DeviceId := evStartRequestData.DeviceId);
IF fbCheckReady.bReady THEN
   bMoveBwdDone := TRUE;
END_IF;

@F
@Acb @RT(19)AStopMovementFwdBwd @F @T @RT(2)P0 @RT(0) @F @F @T @TL(2)
aStopMovementBwd();

@F

@AltBranch @RT(3)alt @F 2
@TransSeq @RT(4)tseq @F 1
@Trans @RT(12)TMoveBwdDone @F @T @F @F @T @T @TL(2)
bMoveBwdDone

@RT(12)TMoveBwdDone @F

@TransSeq @RT(4)tseq @F 4
@Trans @RT(12)TStopMoveBwd @F @T @F @F @T @F @TL(6)
sv_GlobalIdentMaxSpeedStatus.Status = tnCalibState_Aborted OR
sv_GlobalIdentMaxSpeedStatus.Status = tnCalibState_None
OR sv_iPendingAlarms <> 0
OR mActMovement^.bRedo = FALSE

@RT(12)TStopMoveBwd @F
@Step @RT(13)S_StopMoveBwd @F @F @T @F @RT(0) @F
@AcbCont @RT(7)unnamed @F 1
@Acb @RT(12)AStopMoveBwd @F @T @RT(1)P @RT(0) @F @F @T @TL(2)
aStopMovementError(sMovementName := CONCAT(sMoveName, ' max ident Fwd: Bwd to start position'));

@F

@Trans @RT(7)TReset2 @F @T @F @F @T @T @TL(2)
TRUE

@RT(7)TReset2 @F
@Goto @RT(7)S_RESET @F @F

@Step @RT(23)S_CHECK_ALARMS_RETRYFWD @F @F @F @F @RT(0) @F
@AcbCont @RT(7)unnamed @F 0

@AltBranch @RT(3)alt @F 2
@TransSeq @RT(4)tseq @F 1
@Trans @RT(9)TRetryFwd @F @T @F @F @T @T @TL(2)
S_CHECK_ALARMS_RETRYFWD.T > T#1s

@RT(9)TRetryFwd @F

@TransSeq @RT(4)tseq @F 2
@Trans @RT(14)TStopIdentFwd4 @F @T @F @F @T @F @TL(2)
sv_iPendingAlarms <> 0

@RT(14)TStopIdentFwd4 @F
@Goto @RT(13)S_StopMoveBwd @F @F

@Goto @RT(11)S_CALIB_FWD @F @F

@Step @RT(25)S_InitStartMovementBwdFwd @F @F @F @F @RT(0) @F
@AcbCont @RT(7)unnamed @F 3
@Acb @RT(24)AInitStartMovementBwdFwd @F @T @RT(1)P @RT(0) @F @F @T @TL(4)
bMoveFwdDone := FALSE;
miErrorNo := cIdentSpeedMaxFwdInit;
aStartMovementFwd();

@F
@Acb @RT(29)ACheckInitMovementBwdFwdReady @F @T @RT(1)N @RT(0) @F @F @T @TL(5)
fbCheckReady(DeviceId := evStartRequestData.DeviceId);
IF fbCheckReady.bReady THEN
   bMoveFwdDone := TRUE;
END_IF;

@F
@Acb @RT(23)AStopInitMovementBwdFwd @F @T @RT(2)P0 @RT(0) @F @F @T @TL(2)
aStopMovementFwd();

@F

@AltBranch @RT(3)alt @F 2
@TransSeq @RT(4)tseq @F 1
@Trans @RT(7)Trans35 @F @T @F @F @T @T @TL(2)
bMoveFwdDone

@RT(7)Trans35 @F

@TransSeq @RT(4)tseq @F 4
@Trans @RT(16)TStopInitMoveFwd @F @T @F @F @T @F @TL(5)
sv_GlobalIdentMaxSpeedStatus.Status = tnCalibState_Aborted OR
sv_GlobalIdentMaxSpeedStatus.Status = tnCalibState_None
OR sv_iPendingAlarms <> 0
OR mActMovement^.bRedo = FALSE

@RT(16)TStopInitMoveFwd @F
@Step @RT(17)S_StopInitMoveFwd @F @F @T @F @RT(0) @F
@AcbCont @RT(7)unnamed @F 1
@Acb @RT(16)AStopInitMoveFwd @F @T @RT(1)P @RT(0) @F @F @T @TL(2)
aStopMovementError(sMovementName := CONCAT(sMoveName, ' max ident Bwd: Fwd to initial position'));

@F

@Trans @RT(17)TResetInitMoveFwd @F @T @F @F @T @T @TL(2)
TRUE

@RT(17)TResetInitMoveFwd @F
@Goto @RT(7)S_RESET @F @F

@Step @RT(23)S_CHECK_ALARMS_STARTBWD @F @F @F @F @RT(0) @F
@AcbCont @RT(7)unnamed @F 0

@AltBranch @RT(3)alt @F 2
@TransSeq @RT(4)tseq @F 1
@Trans @RT(13)TStartInitBwd @F @T @F @F @T @T @TL(2)
S_CHECK_ALARMS_STARTBWD.T > T#100ms

@RT(13)TStartInitBwd @F

@TransSeq @RT(4)tseq @F 2
@Trans @RT(14)TStopIdentFwd3 @F @T @F @F @T @F @TL(2)
sv_iPendingAlarms <> 0

@RT(14)TStopIdentFwd3 @F
@Goto @RT(17)S_StopInitMoveFwd @F @F

@Step @RT(15)S_INITCALIB_BWD @F @F @F @F @RT(0) @F
@AcbCont @RT(7)unnamed @F 1
@Acb @RT(13)AInitCalibBwd @F @T @RT(1)P @RT(0) @F @F @T @TL(19)
iFileCounter := 1;
IF (CHECK_REF(mActMovement^.prSizeFactorBwd^)) THEN
   IF (mActMovement^.prSizeFactorBwd^ > 0.0) THEN
      rVelocitSizeFactor := mActMovement^.prSizeFactorBwd^;
   END_IF;
ELSE
   rVelocitSizeFactor := 1.0;
END_IF;
rRefSpeedLimit := mActMovement^.prVelocityLimitBwd^;
rMaxPressureLimit := mActMovement^.prMaxPressureBwd^;
IF CHECK_REF(mActMovement^.prMaxPressureBwdHydr^) THEN
   rMaxRefPressureLimit := mActMovement^.prMaxPressureBwdHydr^;
ELSE
   rMaxRefPressureLimit := mActMovement^.prMaxPressureFwd^;
END_IF;

dummy := Print('Calib max speed %s Bwd started', sMoveName);

@F

@Trans @RT(13)TInitCalibBwd @F @T @F @F @T @T @TL(2)
S_INITCALIB_BWD.T>T#1s

@RT(13)TInitCalibBwd @F
@Step @RT(11)S_CALIB_BWD @F @F @T @F @RT(0) @F
@AcbCont @RT(7)unnamed @F 4
@Acb @RT(11)ADoCalibBwd @F @T @RT(1)P @RT(0) @F @F @T @TL(50)
ConstVis := mActMovement^.pConstBwdVis^;

mActMovement^.pConstBwdVis^.Velocity.Output.rOutputValue := rRefSpeedLimit * rVelocitSizeFactor;
mActMovement^.pConstBwdVis^.Velocity.rMinOutput := 0.0;
mActMovement^.pConstBwdVis^.Pressure.Output.rOutputValue := MAX(mActMovement^.pConstBwdVis^.Pressure.Output.rOutputValue, rMaxPressureLimit);
mActMovement^.pConstBwdVis^.Pressure.Output.rRamp := MAX(1.0e9,ConstVis.Pressure.Output.rRamp);
IF mActMovement^.bPositionIncreasingFwd THEN
   mActMovement^.prIdentPosition^ := mActMovement^.prStroke^ * mrMinPositionFactor;
   mrMaxLimitPosition := rStartFactor * mActMovement^.prIdentPosition^ + (1.0 - rStartFactor) * mActMovement^.prPosition^;
   rMinStopRamp := rRefSpeedLimit / ABS(mActMovement^.prIdentPosition^ - mActMovement^.prPosition^);
   IF (mActMovement^.prPosition^ - mActMovement^.prIdentPosition^) > 0.0 THEN
      rMinStopRamp := rMinStrokeFactor * rRefSpeedLimit * rRefSpeedLimit / ABS(mActMovement^.prIdentPosition^ - mActMovement^.prPosition^);
   ELSE
      rMinStopRamp := 0.0;
   END_IF;
   mActMovement^.prStopRamp^ := MAX(mActMovement^.pConstBwdVis^.Velocity.Output.rRamp, rMinStopRamp);
   mrMinLimitPosition := mActMovement^.prIdentPosition^;
ELSE
   mActMovement^.prIdentPosition^ := mActMovement^.prStroke^ * mrMaxPositionFactor;
   mrMinLimitPosition := rStartFactor * mActMovement^.prPosition^ + (1.0 - rStartFactor) * mActMovement^.prIdentPosition^;
   IF (mActMovement^.prIdentPosition^ - mActMovement^.prPosition^) > 0.0 THEN
      rMinStopRamp := rMinStrokeFactor * rRefSpeedLimit * rRefSpeedLimit / ABS(mActMovement^.prIdentPosition^ - mActMovement^.prPosition^);
   ELSE
      rMinStopRamp := 0.0;
   END_IF;
   mActMovement^.prStopRamp^ := MAX(mActMovement^.pConstBwdVis^.Velocity.Output.rRamp, rMinStopRamp);
   mrMaxLimitPosition := mActMovement^.prIdentPosition^;
END_IF;
mActMovement^.pbMoveIdent^ := TRUE;

bMoveIdentDone := FALSE;

mrRefVelocity := rRefSpeedLimit;
mrRefPressure := rMaxRefPressureLimit;
mbRestartMeas := TRUE;

IF bDelayTimeOffFwdLinked THEN
   mActMovement^.pdDelayTimeOffFwd^ := MAX(mActMovement^.pdDelayTimeOffFwd^, dMinDelayTimeOff);
END_IF;
IF bDelayTimeOffBwdLinked THEN
   mActMovement^.pdDelayTimeOffBwd^ := MAX(mActMovement^.pdDelayTimeOffBwd^, dMinDelayTimeOff);
END_IF;

aStartMeasurement();

sWriteSpeedLimit := REAL_TO_STRING(rRefSpeedLimit);
dummy := Print('Calib max output: act. max speed: %s', sWriteSpeedLimit);
miErrorNo := cIdentSpeedMaxBwdIdent;

@F
@Acb @RT(17)AStartMovementBwd @F @T @RT(1)P @RT(0) @F @F @T @TL(9)
evStartRequestData.DeviceId := mActMovement^.DeviceId;
evStartRequestData.MoveDir := cMoveBwd;
IF mActMovement^.MoveId > cMoveNone THEN
   evStartRequestData.MoveId := cMoveDecompAftPlast;
ELSE
   evStartRequestData.MoveId := cMoveBwd;
END_IF;
SET_EVENT(evStartRequest, evStartRequestData);

@F
@Acb @RT(25)ACheckActMovementBwdReady @F @T @RT(1)N @RT(0) @F @F @T @TL(5)
fbCheckReady(DeviceId := evStartRequestData.DeviceId);
IF fbCheckReady.bReady THEN
   bMoveIdentDone := TRUE;
END_IF;

@F
@Acb @RT(16)AStopMovementBwd @F @T @RT(2)P0 @RT(0) @F @F @T @TL(15)
aStopMeasurement();
aStopMovementBwd();

mActMovement^.pConstBwdVis^ := ConstVis;
mActMovement^.prStopRamp^ := 0.0;

IF bDelayTimeOffFwdLinked THEN
   mActMovement^.pdDelayTimeOffFwd^ := dDelayTimeOffFwd;
END_IF;
IF bDelayTimeOffBwdLinked THEN
   mActMovement^.pdDelayTimeOffBwd^ := dDelayTimeOffBwd;
END_IF;

@F

@AltBranch @RT(3)alt @F 2
@TransSeq @RT(4)tseq @F 1
@Trans @RT(7)Trans14 @F @T @F @F @T @T @TL(2)
bMoveIdentDone

@RT(7)Trans14 @F

@TransSeq @RT(4)tseq @F 4
@Trans @RT(13)TStopCalibBwd @F @T @F @F @T @F @TL(5)
sv_GlobalIdentMaxSpeedStatus.Status = tnCalibState_Aborted OR
sv_GlobalIdentMaxSpeedStatus.Status = tnCalibState_None
OR sv_iPendingAlarms <> 0
OR mActMovement^.bRedo = FALSE

@RT(13)TStopCalibBwd @F
@Step @RT(14)S_StopCalibBwd @F @F @T @F @RT(0) @F
@AcbCont @RT(7)unnamed @F 1
@Acb @RT(13)AStopCalibBwd @F @T @RT(1)P @RT(0) @F @F @T @TL(2)
aStopMovementError(sMovementName := CONCAT(sMoveName, ' max ident Bwd'));

@F

@Trans @RT(14)TResetCalibBwd @F @T @F @F @T @F @TL(2)
TRUE

@RT(14)TResetCalibBwd @F
@Goto @RT(7)S_RESET @F @F

@Step @RT(18)S_CHECK_ALARMS_BWD @F @F @F @F @RT(0) @F
@AcbCont @RT(7)unnamed @F 0

@AltBranch @RT(3)alt @F 2
@TransSeq @RT(4)tseq @F 1
@Trans @RT(14)TStartWriteBwd @F @T @F @F @T @T @TL(2)
S_CHECK_ALARMS_BWD.T > T#100ms

@RT(14)TStartWriteBwd @F

@TransSeq @RT(4)tseq @F 2
@Trans @RT(14)TStopCalibBwd2 @F @T @F @F @T @F @TL(2)
sv_iPendingAlarms <> 0

@RT(14)TStopCalibBwd2 @F
@Goto @RT(14)S_StopCalibBwd @F @F

@Step @RT(11)S_WRITE_BWD @F @F @F @F @RT(0) @F
@AcbCont @RT(7)unnamed @F 1
@Acb @RT(9)AWriteBwd @F @T @RT(1)P @RT(0) @F @F @T @TL(11)
abSpeedMeasure.aGetMaxValues(rMaxSpeed => mrMaxVelocity,
                             rMaxPressure => mrMaxPressure,
                             bPressureLimitReached => mbPressureLimitReached,
                             bSpeedLimitReached => mbVelocityLimitReached);
sFileName := CONCAT(sMoveName,"_MAXSPEED_BWD_");
aWriteLog(sFileName := sFileName,
          iFileCounter := iFileCounter,
          bDeleteFiles := TRUE);
iFileCounter := iFileCounter + 1;

@F

@Trans @RT(9)TWriteBwd @F @T @F @F @T @T @TL(2)
mbLogFileSaved

@RT(9)TWriteBwd @F
@Step @RT(20)S_CHECK_MAXSPEED_BWD @F @F @F @F @RT(0) @F
@AcbCont @RT(7)unnamed @F 1
@Acb @RT(17)ACheckMaxSpeedBwd @F @T @RT(1)P @RT(0) @F @F @T @TL(18)
aCalcMaxSpeedOutput(rMaxSpeedLimit := mActMovement^.prVelocityLimitBwd^,
                    rActSpeedLimit := rRefSpeedLimit,
                    rActMaxSpeed := abSpeedMeasure.aGetMaxValues.rMaxSpeed,
                    bPresLimitReached := abSpeedMeasure.aGetMaxValues.bPressureLimitReached,
                    bUsePressureMode := (mrMaxPressure > 0.0));
bMaxBwdDetected := aCalcMaxSpeedOutput.bMaxDetected;
IF (bMaxBwdDetected) THEN
   rSpeedLimitBwd := rRefSpeedLimit;
   dummy := Print('Calib max output %s Bwd finished: max speed bwd = %f$N', sMoveName, rSpeedLimitBwd);
ELSE
   IF abSpeedMeasure.aGetMaxValues.bPressureLimitReached THEN
      sWriteSpeedLimit := REAL_TO_STRING(rRefSpeedLimit);
      dummy := Print('Calib max output: pressure limit reached with act. max speed %s', sWriteSpeedLimit);
   END_IF;
   bMaxBwdRetry := TRUE;
   rRefSpeedLimit := aCalcMaxSpeedOutput.rRefSpeed;
END_IF;

@F

@AltBranch @RT(3)alt @F 2
@TransSeq @RT(4)tseq @F 1
@Trans @RT(15)TMaxBwdDetected @F @T @F @F @T @T @TL(2)
bMaxBwdDetected

@RT(15)TMaxBwdDetected @F

@TransSeq @RT(4)tseq @F 6
@Trans @RT(12)TMaxBwdRetry @F @T @F @F @T @T @TL(2)
bMaxBwdRetry

@RT(12)TMaxBwdRetry @F
@Step @RT(13)S_MaxBwdRetry @F @F @F @F @RT(0) @F
@AcbCont @RT(7)unnamed @F 3
@Acb @RT(20)AStartMovementBwdFwd @F @T @RT(1)P @RT(0) @F @F @T @TL(4)
bMoveFwdDone := FALSE;
miErrorNo := cIdentSpeedMaxBwdStart;
aStartMovementFwd();

@F
@Acb @RT(28)ACheckActMovementBwdFwdReady @F @T @RT(1)N @RT(0) @F @F @T @TL(5)
fbCheckReady(DeviceId := evStartRequestData.DeviceId);
IF fbCheckReady.bReady THEN
   bMoveFwdDone := TRUE;
END_IF;

@F
@Acb @RT(19)AStopMovementBwdFwd @F @T @RT(2)P0 @RT(0) @F @F @T @TL(2)
aStopMovementFwd();

@F

@AltBranch @RT(3)alt @F 2
@TransSeq @RT(4)tseq @F 1
@Trans @RT(12)TMoveFwdDone @F @T @F @F @T @T @TL(2)
bMoveFwdDone

@RT(12)TMoveFwdDone @F

@TransSeq @RT(4)tseq @F 4
@Trans @RT(12)TStopMoveFwd @F @T @F @F @T @F @TL(6)
sv_GlobalIdentMaxSpeedStatus.Status = tnCalibState_Aborted OR
sv_GlobalIdentMaxSpeedStatus.Status = tnCalibState_None
OR sv_iPendingAlarms <> 0
OR mActMovement^.bRedo = FALSE

@RT(12)TStopMoveFwd @F
@Step @RT(13)S_StopMoveFwd @F @F @T @F @RT(0) @F
@AcbCont @RT(7)unnamed @F 1
@Acb @RT(12)AStopMoveFwd @F @T @RT(1)P @RT(0) @F @F @T @TL(2)
aStopMovementError(sMovementName := CONCAT(sMoveName, ' max ident Bwd: Fwd to start position'));
